# B&R Automation Studio project TD52 (part 98)

#### MsgEXCyclic.st
```iecst
(*******************************************************************************
MsgEX	 			 alarms, messages MM_EX

This code is confidential and proprietary to the INNIO Company.
It may not be used in any form, or reproduced in any manner,
without written permission of the INNIO Company.
Copyright, INNIO Company, 2025

Customized modifications: -
------------------------

History:
-------
V3.99.0	04.06.2012	lettenb.	new
		20.03.2013				para.cleanup
		23.04.2013				reset OUT_EX.tEX2AB.bGnlWarning added
		16.05.2013				3349,3580,3581,3582 added from V3.30.x
		23.05.2013				2847,2848 added
		24.05.2013				reset OUT_xx.txx2AB.bGnlTripx changed
		28.05.2013				2622,2623 for 424tstc added
		04.06.2013				1163,1171 var.names changed(EGbHE -> EGaTC)
								1172 limit var.changed, bugfix
		23.07.2013				2576,2577 enabled if sensor active
		17.01.2014				3366,3417 added, 1165 disabled (exh.gas scav. after engine stop)
V4.00.0	26.02.2014				logger entries added
V4.00.1	09.04.2014				3417 disabled for engines without EGScav
V4.00.2	14.05.2014				1172 KK_AUF AND BTRB added, ton 0s->120s (anforderung requisition/poppe,a_v3500)
		27.05.2014				1172 KK_AUF -> OUT_EX.EG_BoVaOpened (universal for combi valves)
		23.06.2014				2098 logic in case of Para.bSel_EGVa_Combi separated, bugfix
		08.08.2014				3417 IN_EX.bMsg1078 added, to avoid alarm in case of signal failure
V4.00.3 21.01.2015 lettenb.		2655-2664 added(Gen2 engine controller)
		11.02.2015				1165,3366 prepared FOR blackstart,
								3510 logic corr.(bugfix)
								1163 enable with IN_VE.tPB2MM.bSys_Run
								1273-1280 added
V4.03.0 27.07.2015 Plattner		2743 - 2748 & 3397 added. differential pressure exhaust gas cooler and filter limits and msf
								1288 - 1291 added operations message from CO2 flap
        05.08.2015 Stary        added 3394+3395 & 3490+3491
		14.07.2016 lettenb.		3491 xGR_MAXR_T_EGaHE2_LimHi_Warn: Ai+Para changed, 3394,3395,3490,3491 TON 0->2s, double 3395 removed, bugfix
		22.09.2016 lettenb.		1291 NOT added, bugfix
		04.10.2016				2793 added, FC monitoring
		09.02.2017				3417 trip prio corr. 3 -> 4
V4.05.0 21.03.2017 lettenb.     3100 disabled for 920, SWAT920/2
		28.06.2017				2847,2848 N2 gas valve open/closed changed, bugfix
		12.07.2017 Messner		A2315, W2468, W2469 added and W3417 para added
		09.10.2017 Weitzer		3100 enable for 920 again! Increase time delay from 2s TO 120s. SWAT920/x
		02.08.2017				2847,2848 N2 valves open/closed changed, synch.acc.VIS, bu09
		04.12.2017 Messner		Oxidation catalyst added
								Old KAT Disabled: A1045, A1069; W1161, W1162,  W1169, W1170, W1174, W2112;
								New OXIcat Added: A2319, A2320; W2494, W2495, W2496, W2497, W2498, W2499, W2500;
		22.05.2017	TinelloM	SCR deleted
		20.12.2017	lettenb.	A3397 prio: 4->3, bugfix
		02.01.2017	lettenb.	3417 disabled for 920 with common gas train(main and prechamber)(not for ACEA,sky,rosenheim,stapelfeld)
		18.01.2018				2310,2311,2312,2313 added, 1171,2546,2547:Para.rT_EGaTC_HyHi removed(burkhart)
		22.01.2018	lettenb.	1163,1164,2793 bSys_Run -> bParaSetupOk to avoid message at plc startup
V4.05.1 19.03.2018	lettenb.    2320,2500 delay 1s added to avoid alarm with siganl failure, bugfix
V4.07.0 26.04.2018	lettenb.	9215 added, 1165 enabled for BR9, 3366 disabled for BR9, SWAT920/5
		08.10.2018	lettenb.	3214, :bOMSS... removed, signal failure active in stop-mode
		31.10.2018	lettenb.	2321,2322 added, (burkhart)
		03.12.2018	lettenb.	1165,3366,1279,1280 NoScavFan added, bugfix for option N2 scav.without scav.fan
		14.01.2019	Schmid		A2340+W9249 added, W2498+W2497 deactivated, "exhaust gas pressure fast" fully replaces "OXIcat inlet pressure fast"
		18.03.2019	lettenb.	2497,2498 cleanup unused code
		13.06.2019	lettenb.	1171,2310,2311,2546,2547: MM2VIS.bMsg2312/2313/2322 added to avoid hi-alarm with MS, bugfix
		03.10.2019	lettenb.	9310 added, 2319 disabled, OXIcat monitoring, bu
V4.09.0	02.08.2019	lettenb.	2337,2338,9305-9308: temperature exhaust gas pressure relief valve 1/2 added
		13.07.2020	lettenb.	2496 time delay 60s added, bu
V4.11.0 04.03.2021	lettenb.	9347,9348 added, exhaust gas flap monitoring
V4.12.0	19.12.2022	Perktold	added comments for sr-code (EN 13849-1 / 4.6.3) for A1092,A2315 & W3528
V4.13.0	19.10.2023	Heim Markus	add A2374 (defined as safety critical no remote reset possible (riskclass 10)
V4.14.0	16.10.2024	VighM		W9249 set by bad signal quality, delay cleanup.
V4.14.0	06.11.2024	Theobald	At alarm 1092 only temperature sensor cause trip while the engine is running and at alarm 3366 there is no trip during engine operation.
		25.11.2024	Bacci		T6 Start procedure with purge start (2024-219): scavenging fan removal
V4.25.0	10.07.2025	Tinello	 	SafetyPLC: Disabled W3528 in case of Safety gas backpressure monitoring active

Instructions for use:
--------------------
1) declare alarm with FUNCTION block "Alm"
	declare buffert alarm bit bMsg<message number>

2) use template to create a new alarm,
   substitue 0000 by alarm number and make settings:

	xMsg0000.Enable		:=	TRUE;		enable/disable alarm
	xMsg0000.Set		:=	FALSE;		alarm set condition
	xMsg0000.PT			:=	T#0s;		alarm delay time
	xMsg0000.Prio		:=	1;			alarm priority: 1-3 = trip, 4 = warning
	xMsg0000.RiskClass	:=	3;			risk class for remote alarm reset
	xMsg0000.Reset		:=	FALSE;		FALSE: for all standard alarms	prio 1,2,3 and warnings prio 4
										TRUE : for autoreset alarms

	bMsg0000			:=	xMsg0000.Q;	connect buffert alarm bit for VIS and control
	bMsg0000_Test		:=	xMsg0000.Test; alarm bypass active

3)  expand INIT

4)	include datapoint into OPC configuration for vis

Outstandings:
------------
logic FOR alarm 2622,2623 (424)
W exhaust gas scavenging before next start
(*******************************************************************************)
PROGRAM _CYCLIC

	(* reset general trip *)
	OUT_EX.tEX2AB.bGnlTrip1		:=	FALSE;
	OUT_EX.tEX2AB.bGnlTrip2		:=	FALSE;
	OUT_EX.tEX2AB.bGnlTrip3		:=	FALSE;
	OUT_EX.tEX2AB.bGnlWarning	:=	FALSE;
	OUT_EX.tEX2AB.bTriptype1	:=	FALSE;
	OUT_EX.tEX2AB.bTriptype2	:=	FALSE;
	OUT_EX.tEX2AB.bTriptype3	:=	FALSE;

	(*-------------------------------------------------------------------------*)
	(* A1045 catalyst temperature high (W1174) *) (* Disabled - OXIcat *)
	xMsg1045.Enable	   := FALSE;
	xMsg1045.Set	   := FALSE;
	xMsg1045.PT		   := T#0s;
	xMsg1045.Prio 	   := 2;
	xMsg1045.RiskClass := 4;
	xMsg1045.Reset     := FALSE;
	xMsg1045();
	MM2VIS.bMsg1045    := xMsg1045.Q;

	(* A1046 exhaust gas flap failure (--> W2098) *)
	xMsg1046.Enable	   := FALSE;
	xMsg1046.Set 	   := FALSE;
	xMsg1046.PT		   := T#0s;
	xMsg1046.Prio 	   := 3;
	xMsg1046.RiskClass := 3;
	xMsg1046.Reset     := FALSE;
	xMsg1046();
	MM2VIS.bMsg1046    := xMsg1046.Q;

	(* A1069 catalyst temperature signal failure (W2112) *) (* Disabled - OXIcat *)
	xMsg1069.Enable	   := FALSE;
	xMsg1069.Set 	   := FALSE;
	xMsg1069.PT		   := T#0s;
	xMsg1069.Prio 	   := 3;
	xMsg1069.RiskClass := 2;
	xMsg1069.Reset     := FALSE;
	xMsg1069();
	MM2VIS.bMsg1069    := xMsg1069.Q;

	(********************************************************************************************************************
	Safety-related application software source code (EN 13849-1 / 4.6.3): BEGIN
	*********************************************************************************************************************)

	(* A1092 exhaust gas scavenging valve failure *)
	xMsg1092.Enable	   := TRUE;
	xMsg1092.Set 	   := (T1_STSPKL AND NOT IN_EX.tEng_Run.Do) OR T2_STSPKL;
	xMsg1092.PT		   := T#0s;
	xMsg1092.Prio 	   := 2;
	xMsg1092.RiskClass := 10;
	xMsg1092.Reset     := FALSE;
	xMsg1092();
	MM2VIS.bMsg1092    := xMsg1092.Q;

	(********************************************************************************************************************
	Safety-related application software source code (EN 13849-1 / 4.6.3): END
	*********************************************************************************************************************)

	(* A1104 plate temperature heat exchanger high *)
	xGR_MAXR_T_PlateHE_LimHiHi(In:= IN_EX.tT_PlateHE.Ai, Gw:= Para.rT_PlateHE_LimHiHi, Hy:= Para.rT_PlateHE_HyHi);

	xMsg1104.Enable	   := Para.bT_PlateHE_Active;
	xMsg1104.Set 	   := xGR_MAXR_T_PlateHE_LimHiHi.Q AND IN_EX.tPB2MM.bParaSetupOk AND NOT MM2VIS.bMsg2113;
	xMsg1104.PT		   := T#2s;
	xMsg1104.Prio 	   := 3;
	xMsg1104.RiskClass := 4;
	xMsg1104.Reset     := FALSE;
	xMsg1104();
	MM2VIS.bMsg1104    := xMsg1104.Q;

	(* A1106 plate temperature heat exchanger signal failure(--> W2113) *)
	xMsg1106.Enable	   := Para.bT_PlateHE_Active AND FALSE;
	xMsg1106.Set 	   := NOT IN_EX.tT_PlateHE.GoodQual;
	xMsg1106.PT		   := T#0s;
	xMsg1106.Prio 	   := 3;
	xMsg1106.RiskClass := 4;
	xMsg1106.Reset     := FALSE;
	xMsg1106();
	MM2VIS.bMsg1106    := xMsg1106.Q;

	(* W1161 exhaust gas temperature before catalyst signal failure *) (* Disabled - OXIcat *)
	xMsg1161.Enable	   := FALSE;
	xMsg1161.Set 	   := FALSE;
	xMsg1161.PT		   := T#0s;
	xMsg1161.Prio 	   := 4;
	xMsg1161.RiskClass := 4;
	xMsg1161.Reset     := FALSE;
	xMsg1161();
	MM2VIS.bMsg1161    := xMsg1161.Q;

	(* W1162 exhaust gas temperature after catalyst signal failure *) (* Disabled - OXIcat *)
	xMsg1162.Enable	   := FALSE;
	xMsg1162.Set 	   := FALSE;
	xMsg1162.PT		   := T#0s;
	xMsg1162.Prio 	   := 4;
	xMsg1162.RiskClass := 4;
	xMsg1162.Reset     := FALSE;
	xMsg1162();
	MM2VIS.bMsg1162    := xMsg1162.Q;

	(* W1163 (A2322) exhaust gas temperature after turbo charger signal failure *)
	xMsg1163.Enable	   := Para.bT_EGaTC_Active AND IN_EX.tPB2MM.bParaSetupOk;
	xMsg1163.Set 	   := NOT IN_EX.tT_EGaTC.GoodQual AND NOT Para.bT_EGaLPTC_HiTrip;
	xMsg1163.PT		   := T#0s;
	xMsg1163.Prio 	   := 4;
	xMsg1163.RiskClass := 4;
	xMsg1163.Reset     := FALSE;
	xMsg1163();
	MM2VIS.bMsg1163    := xMsg1163.Q;

	(* W1164 exhaust gas temperature after heat exchanger signal failure *)
	xMsg1164.Enable	   := Para.bT_EGaHE_Active AND IN_EX.tPB2MM.bParaSetupOk;
	xMsg1164.Set 	   := NOT IN_EX.tT_EGaHE.GoodQual;
	xMsg1164.PT		   := T#0s;
	xMsg1164.Prio 	   := 4;
	xMsg1164.RiskClass := 4;
	xMsg1164.Reset     := FALSE;
	xMsg1164();
	MM2VIS.bMsg1164    := xMsg1164.Q;

   (* W1165 exhaust gas scavenging fan failure (A3366) *)
	xTOF_EngDemEPS(IN:= IN_EX.bEng_Dem_EPS AND NOT IN_EX.tGCB_On.Di, PT:= T#60s);
	bNoMon4BlackStart := xTOF_EngDemEPS.Q AND IN_EX.bEng_Dem_EPS; //T14

	xMsg1165.Enable	   := xEngType.Type9;//SWAT920/5
	xMsg1165.Set 	   :=	OUT_EX.tScavFanCoOn.Do
					AND NOT bNoMon4BlackStart
					AND(   (NOT xEngType.Type9 AND NOT IN_EX.tScavFanOp.Di AND NOT NoScavFan)
						OR (    xEngType.Type9 AND    (IN_EX.tScavFanFC_P_Lo.Di OR NOT IN_EX.tScavFanFC_Rdy.Di)));
	xMsg1165.PT		   := T#10s;
	xMsg1165.Prio 	   := 4;
	xMsg1165.RiskClass := 4;
	xMsg1165.Reset     := FALSE;
	xMsg1165();
	MM2VIS.bMsg1165	   := xMsg1165.Q;
	OUT_EX.bMsg1165	   := xMsg1165.Q;//SWAT920/5

	(* W1169 exhaust gas temperature before catalyst high *) (* Disabled - OXIcat *)
	xMsg1169.Enable	   := FALSE;
	xMsg1169.Set 	   := FALSE;
	xMsg1169.PT		   := T#2s;
	xMsg1169.Prio 	   := 4;
	xMsg1169.RiskClass := 4;
	xMsg1169.Reset     := FALSE;
	xMsg1169();
	MM2VIS.bMsg1169    := xMsg1169.Q;

	(* W1170 exhaust gas temperature after catalyst high *) (* Disabled - OXIcat *)
	xMsg1170.Enable	   := FALSE;
	xMsg1170.Set 	   := FALSE;
	xMsg1170.PT		   := T#2s;
	xMsg1170.Prio 	   := 4;
	xMsg1170.RiskClass := 4;
	xMsg1170.Reset     := FALSE;
	xMsg1170();
	MM2VIS.bMsg1170    := xMsg1170.Q;

	(* W1171 (A2321) exhaust gas temperature after turbo charger high *)
	xGR_MAXR_T_EGaTC_LimHi(In:= IN_EX.tT_EGaTC.Ai, Gw:= Para.rT_EGaTC_LimHi, Hy:= 5.0);

	xMsg1171.Enable	   := Para.bT_EGaTC_Active;
	xMsg1171.Set 	   := xGR_MAXR_T_EGaTC_LimHi.Q AND IN_EX.tPB2MM.bParaSetupOk AND NOT MM2VIS.bMsg1163 AND NOT MM2VIS.bMsg2322;
	xMsg1171.PT		   := T#2s;
	xMsg1171.Prio 	   := 4;
	xMsg1171.RiskClass := 4;
	xMsg1171.Reset     := FALSE;
	xMsg1171();
	MM2VIS.bMsg1171    := xMsg1171.Q;

	(* W1172 exhaust gas temperature after heat exchanger high *)
	xGR_MAXR_T_EGaHE_LimHi(In:= IN_EX.tT_EGaHE.Ai, Gw:= Para.rT_EGaHE_LimHi, Hy:= Para.rT_EGaHE_HyHi);

	xMsg1172.Enable	   := Para.bT_EGaHE_Active;
	xMsg1172.Set 	   := xGR_MAXR_T_EGaHE_LimHi.Q AND IN_EX.tPB2MM.bParaSetupOk AND NOT MM2VIS.bMsg1164
					  AND OUT_EX.bEG_BoVaOpened AND IN_EX.tEng_Run.Do;
	xMsg1172.PT		   := T#120s;
	xMsg1172.Prio 	   := 4;
	xMsg1172.RiskClass := 4;
	xMsg1172.Reset     := FALSE;
	xMsg1172();
	MM2VIS.bMsg1172    := xMsg1172.Q;

	(* W1173 plate temperature heat exchanger high *)
	xGR_MAXR_T_PlateHE_LimHi(In:= IN_EX.tT_PlateHE.Ai, Gw:= Para.rT_PlateHE_LimHi, Hy:= Para.rT_PlateHE_HyHi);

	xMsg1173.Enable	   := Para.bT_PlateHE_Active;
	xMsg1173.Set 	   := xGR_MAXR_T_PlateHE_LimHi.Q AND IN_EX.tPB2MM.bParaSetupOk AND NOT MM2VIS.bMsg2113;
	xMsg1173.PT		   := T#2s;
	xMsg1173.Prio 	   := 4;
	xMsg1173.RiskClass := 4;
	xMsg1173.Reset     := FALSE;
	xMsg1173();
	MM2VIS.bMsg1173    := xMsg1173.Q;

	(* W1174 catalyst temperatur high (A1045) *) (* Disabled - OXIcat *)
	xMsg1174.Enable	   := FALSE;
	xMsg1174.Set 	   := FALSE;
	xMsg1174.PT		   := T#2s;
	xMsg1174.Prio 	   := 4;
	xMsg1174.RiskClass := 4;
	xMsg1174.Reset     := FALSE;
	xMsg1174();
	MM2VIS.bMsg1174    := xMsg1174.Q;

	(* W2098 exhaust gas flap failure *)
	IF Para.bSel_EGVa_Combi THEN
		xTON_2098a(IN:= (NOT IN_EX.tEG_ByVaOpened.Di AND NOT IN_EX.tEG_ByVaClosed.Di AND(B_BKAUF OR B_BKZU)), PT:= T#35s);
	ELSE
		xTON_2098a(IN:= (NOT IN_EX.tEG_ByVaOpened.Di AND NOT IN_EX.tEG_ByVaClosed.Di AND(B_BKAUF OR B_BKZU))
					 OR (NOT IN_EX.tEG_BoVaOpened.Di AND NOT IN_EX.tEG_BoVaClosed.Di AND(B_KKAUF OR B_KKZU)), PT:= T#35s);
	END_IF;
	xTON_2098b(IN:=  NOT IN_EX.tEG_BoVaFailure.Di OR NOT IN_EX.tEG_ByVaFailure.Di, PT:= T#2s);

	xMsg2098.Enable	   := TRUE;
	xMsg2098.Set 	   := xTON_2098a.Q OR xTON_2098b.Q OR (NOT Para.bSel_EGVa_Combi AND NOT IN_EX.tEG_ByVaOpened.Di AND NOT IN_EX.tEG_BoVaOpened.Di);
	xMsg2098.PT		   := T#0s;
	xMsg2098.Prio 	   := 4;
	xMsg2098.RiskClass := 4;
	xMsg2098.Reset     := FALSE;
	xMsg2098();
	MM2VIS.bMsg2098    := xMsg2098.Q;

	(* W2112 catalyst temperature signal failure (A1069) *) (* Disabled - OXIcat *)
	xMsg2112.Enable	   := FALSE;
	xMsg2112.Set 	   := FALSE;
	xMsg2112.PT		   := T#0s;
	xMsg2112.Prio 	   := 4;
	xMsg2112.RiskClass := 4;
	xMsg2112.Reset     := FALSE;
	xMsg2112();
	MM2VIS.bMsg2112    := xMsg2112.Q;

	(* W2113 plate temperature heat exchanger signal failure (A1106) *)
	xMsg2113.Enable	   := Para.bT_PlateHE_Active;
	xMsg2113.Set 	   := NOT IN_EX.tT_PlateHE.GoodQual;
	xMsg2113.PT		   := T#0s;
	xMsg2113.Prio 	   := 4;
	xMsg2113.RiskClass := 4;
	xMsg2113.Reset     := FALSE;
	xMsg2113();
	MM2VIS.bMsg2113    := xMsg2113.Q;

	(* A2310 (W2546) exhaust gas temperature after low pressure turbo charger A high *)(* M.02-TI-168, M.02-TI-001 *)
	xMsg2310.Enable	   := Para.bT_EGaLPTC_A_Active AND Para.bT_EGaLPTC_HiTrip;
	xMsg2310.Set 	   := IN_EX.tPB2MM.bParaSetupOk AND (IN_EX.tT_EGaLPTC_A.Ai > Para.rT_EGaTC_LimHiHi) AND NOT MM2VIS.bMsg2312;
	xMsg2310.PT		   := Para.tiEGaTC_LimHiHi;
	xMsg2310.Prio 	   := 2;
	xMsg2310.RiskClass := 4;
	xMsg2310.Reset     := FALSE;
	xMsg2310();
	MM2VIS.bMsg2310    := xMsg2310.Q;

	(* A2311 (W2547) exhaust gas temperature after low pressure turbo charger B high *)(* M.02-TI-268, M.02-TI-002 *)
	xMsg2311.Enable	   := Para.bT_EGaLPTC_B_Active AND Para.bT_EGaLPTC_HiTrip;
	xMsg2311.Set 	   := IN_EX.tPB2MM.bParaSetupOk AND (IN_EX.tT_EGaLPTC_B.Ai > Para.rT_EGaTC_LimHiHi) AND NOT MM2VIS.bMsg2313;
	xMsg2311.PT		   := Para.tiEGaTC_LimHiHi;
	xMsg2311.Prio 	   := 2;
	xMsg2311.RiskClass := 4;
	xMsg2311.Reset     := FALSE;
	xMsg2311();
	MM2VIS.bMsg2311    := xMsg2311.Q;

	(* A2312 (W2549) exhaust gas temperature after low pressure turbo charger A signal failure *)(* M.02-TI-168, M.02-TI-001 *)
	xMsg2312.Enable	   := Para.bT_EGaLPTC_A_Active AND Para.bT_EGaLPTC_HiTrip;
	xMsg2312.Set 	   := IN_EX.tPB2MM.bParaSetupOk AND NOT IN_EX.tT_EGaLPTC_A.GoodQual;
	xMsg2312.PT		   := T#0s;
	xMsg2312.Prio 	   := 2;
	xMsg2312.RiskClass := 4;
	xMsg2312.Reset     := FALSE;
	xMsg2312();
	MM2VIS.bMsg2312    := xMsg2312.Q;

	(* A2313 (W2551) exhaust gas temperature after low pressure turbo charger B signal failure *)(* M.02-TI-268, M.02-TI-002 *)
	xMsg2313.Enable	   := Para.bT_EGaLPTC_B_Active AND Para.bT_EGaLPTC_HiTrip;
	xMsg2313.Set 	   := IN_EX.tPB2MM.bParaSetupOk AND NOT IN_EX.tT_EGaLPTC_B.GoodQual;
	xMsg2313.PT		   := T#0s;
	xMsg2313.Prio 	   := 2;
	xMsg2313.RiskClass := 4;
	xMsg2313.Reset     := FALSE;
	xMsg2313();
	MM2VIS.bMsg2313    := xMsg2313.Q;

	(********************************************************************************************************************
	Safety-related application software source code (EN 13849-1 / 4.6.3): BEGIN
	*********************************************************************************************************************)

	(* A2315 air temperature before exhaust gas scavening valve maximum *)
	xMsg2315.Enable	   := Para.bT_bScavValve_Active;
	xMsg2315.Set 	   := IN_EX.tPB2MM.bParaSetupOk AND  IN_EX.tT_bScavValve.GoodQual
													AND (IN_EX.rN_EngAct > 0)
													AND (IN_EX.tT_bScavValve.Ai > Para.rT_bScavValve_LimHi);
	xMsg2315.PT		   := T#2s;
	xMsg2315.Prio 	   := 2;
	xMsg2315.RiskClass := 10;
	xMsg2315.Reset     := FALSE;
	xMsg2315();
	MM2VIS.bMsg2315    := xMsg2315.Q;

	(********************************************************************************************************************
	Safety-related application software source code (EN 13849-1 / 4.6.3): END
	*********************************************************************************************************************)

	(* A2319 OXIcat Outlet temperature measurement signal failure *)(* W9310 *)
	xMsg2319.Enable	   := Para.bOXIcat_Exist
					  AND Para.bT_OXIcat_Out_Exist
					  AND FALSE;
	xMsg2319.Set 	   := NOT IN_EX.tT_EGaCat.GoodQual
					  AND (IN_EX.rN_EngAct > 0);
	xMsg2319.PT		   := T#2s;
	xMsg2319.Prio 	   := 3;
	xMsg2319.RiskClass := 4;
	xMsg2319.Reset     := FALSE;
	xMsg2319();
	MM2VIS.bMsg2319    := xMsg2319.Q;

	(* A2320 OXIcat Outlet temperature maximum *)
	xMsg2320.Enable	   := Para.bOXIcat_Exist
					  AND Para.bT_OXIcat_Out_Exist;
	xMsg2320.Set 	   := IN_EX.tT_EGaCat.Ai >= Para.rT_OXIcat_Out_HiHi
					  AND (IN_EX.rN_EngAct > 0)
					  AND IN_EX.tT_EGaCat.GoodQual;
	xMsg2320.PT		   := T#1s;
	xMsg2320.Prio 	   := 2;
	xMsg2320.RiskClass := 4;
	xMsg2320.Reset     := FALSE;
	xMsg2320();
	MM2VIS.bMsg2320    := xMsg2320.Q;

	(* A2321 (W1171) exhaust gas temperature after turbo charger high *)(* M.02-TI-001 *)
	xMsg2321.Enable	   := Para.bT_EGaTC_Active AND Para.bT_EGaLPTC_HiTrip;
	xMsg2321.Set 	   := IN_EX.tPB2MM.bParaSetupOk AND (IN_EX.tT_EGaTC.Ai > Para.rT_EGaTC_LimHiHi) AND NOT MM2VIS.bMsg2322;
	xMsg2321.PT		   := Para.tiEGaTC_LimHiHi;
	xMsg2321.Prio 	   := 2;
	xMsg2321.RiskClass := 4;
	xMsg2321.Reset     := FALSE;
	xMsg2321();
	MM2VIS.bMsg2321    := xMsg2321.Q;

	(* A2322 (W1163) exhaust gas temperature after turbo charger signal failure *)(* M.02-TI-001 *)
	xMsg2322.Enable	   := Para.bT_EGaTC_Active AND Para.bT_EGaLPTC_HiTrip;
	xMsg2322.Set 	   := IN_EX.tPB2MM.bParaSetupOk AND NOT IN_EX.tT_EGaTC.GoodQual;
	xMsg2322.PT		   := T#0s;
	xMsg2322.Prio 	   := 2;
	xMsg2322.RiskClass := 4;
	xMsg2322.Reset     := FALSE;
	xMsg2322();
	MM2VIS.bMsg2322    := xMsg2322.Q;

	(********************************************************************************************************************
	Safety-related application software source code (EN 13849-1 / 4.6.3): BEGIN
	*********************************************************************************************************************)

	(* A2337 (W9305) temperature high exhaust gas pressure relief valve 1 *)(* P.02-TI-039 *)
	xMsg2337.Enable	   := Para.bT_EG_PrReliefVa1_Active;
	xMsg2337.Set 	   := IN_EX.tPB2MM.bParaSetupOk AND(IN_EX.tT_EG_PrReliefVa1.Ai > Para.rT_EG_PrReliefVa_LimHiHi) AND NOT MM2VIS.bMsg9307;
	xMsg2337.PT		   := T#2s;
	xMsg2337.Prio 	   := 3;
	xMsg2337.RiskClass := 10;
	xMsg2337.Reset     := FALSE;
	xMsg2337();
	MM2VIS.bMsg2337    := xMsg2337.Q;

	(* A2338 (W9306) temperature high exhaust gas pressure relief valve 2 *)(* P.02-TI-040 *)
	xMsg2338.Enable	   := Para.bT_EG_PrReliefVa2_Active;
	xMsg2338.Set 	   := IN_EX.tPB2MM.bParaSetupOk AND(IN_EX.tT_EG_PrReliefVa2.Ai > Para.rT_EG_PrReliefVa_LimHiHi) AND NOT MM2VIS.bMsg9308;
	xMsg2338.PT		   := T#2s;
	xMsg2338.Prio 	   := 3;
	xMsg2338.RiskClass := 10;
	xMsg2338.Reset     := FALSE;
	xMsg2338();
	MM2VIS.bMsg2338    := xMsg2338.Q;

	(********************************************************************************************************************
	Safety-related application software source code (EN 13849-1 / 4.6.3): END
	*********************************************************************************************************************)

	(* A2340 Exhaust gas pressure fast maximum (W2498) *)
	xMsg2340.Enable	   := Para.bPr_OXIcat_In_Fast_Exist;
	xMsg2340.Set 	   := bPr_EG_Deflag_Fast
					  AND NOT xTOF_Pr_EG_Deflag_Fast.Q
					  AND ((IN_EX.rN_EngAct > 0) OR IN_EX.bEng_Start) // Prevents continuous setting of the alarm, while bPr_EG_Deflag_Fast remains active
					  AND NOT MM2VIS.bMsg9249;
	xMsg2340.PT		   := T#0s;
	xMsg2340.Prio 	   := 2;
	xMsg2340.RiskClass := 4;
	xMsg2340.Reset     := FALSE;
	xMsg2340();
	MM2VIS.bMsg2340    := xMsg2340.Q;

	(********************************************************************************************************************
	Safety-related application software source code (EN 13849-1 / 4.6.3): BEGIN
	*********************************************************************************************************************)

	(* A2374 Bursting disc triggered (P.02-GS-001/P.02-GS-002)*)
	xMsg2374.Enable	   := IN_EX.tPB2MM.bParaSetupOk;
	xMsg2374.Set 	   := NOT IN_EX.tBurstingDisk1_Ok.Di
					   OR NOT IN_EX.tBurstingDisk2_Ok.Di;
	xMsg2374.PT		   := T#0s;
	xMsg2374.Prio 	   := 2;
	xMsg2374.RiskClass := 10;
	xMsg2374.Reset     := FALSE;
	xMsg2374();
	MM2VIS.bMsg2374    := xMsg2374.Q;

	(********************************************************************************************************************
	Safety-related application software source code (EN 13849-1 / 4.6.3): END
	*********************************************************************************************************************)

	(* W2468 air temperature before exhaust gas scavening valve signal failure *)
	xMsg2468.Enable	   := Para.bT_bScavValve_Active;
	xMsg2468.Set 	   := IN_EX.tPB2MM.bParaSetupOk AND NOT IN_EX.tT_bScavValve.GoodQual;
	xMsg2468.PT		   := T#0s;
	xMsg2468.Prio 	   := 4;
	xMsg2468.RiskClass := 4;
	xMsg2468.Reset     := FALSE;
	xMsg2468();
	MM2VIS.bMsg2468    := xMsg2468.Q;

	(* W2469 air temperature before exhaust gas scavening valve plausibility check *)
	xMsg2469.Enable	   := Para.bT_bScavValve_Active AND FALSE;//SWAT920/5
	xMsg2469.Set 	   := IN_EX.tPB2MM.bParaSetupOk AND bT_bScavValve_PcheckFail;
	xMsg2469.PT		   := T#0s;
	xMsg2469.Prio 	   := 4;
	xMsg2469.RiskClass := 4;
	xMsg2469.Reset     := FALSE;
	xMsg2469();
	MM2VIS.bMsg2469    := xMsg2469.Q;

	(* W2494 OXIcat Inlet pressure measurement signal failure *)
	xMsg2494.Enable	   := Para.bOXIcat_Exist
					  AND Para.bPr_OXIcat_In_Exist;
	xMsg2494.Set 	   := NOT IN_EX.tPr_OXIcat_In.GoodQual
					  AND (IN_EX.rP_Act_Norm_Filt >= 0.50);
	xMsg2494.PT		   := T#60s;
	xMsg2494.Prio 	   := 4;
	xMsg2494.RiskClass := 4;
	xMsg2494.Reset     := FALSE;
	xMsg2494();
	MM2VIS.bMsg2494    := xMsg2494.Q;

	(* W2495 OXIcat Outlet pressure measurement signal failure *)
	xMsg2495.Enable	   := Para.bOXIcat_Exist
					  AND Para.bPr_OXIcat_Out_Exist;
	xMsg2495.Set 	   := NOT IN_EX.tPr_OXIcat_Out.GoodQual
					  AND (IN_EX.rP_Act_Norm_Filt >= 0.50);
	xMsg2495.PT		   := T#60s;
	xMsg2495.Prio 	   := 4;
	xMsg2495.RiskClass := 4;
	xMsg2495.Reset     := FALSE;
	xMsg2495();
	MM2VIS.bMsg2495    := xMsg2495.Q;

	(* W2496 OXIcat Differential pressure minimum *)
	xMsg2496.Enable	   := Para.bOXIcat_Exist
					  AND Para.bPr_OXIcat_In_Exist
					  AND Para.bPr_OXIcat_Out_Exist;
	xMsg2496.Set 	   := MM2VIS.rPr_OXIcat_Diff <= Para.rPR_OXIcat_Diff_Hi
					  AND (IN_EX.rP_Act_Norm_Filt >= 0.50)
					  AND IN_EX.tPr_OXIcat_In.GoodQual
					  AND IN_EX.tPr_OXIcat_Out.GoodQual;
	xMsg2496.PT		   := T#60s;
	xMsg2496.Prio 	   := 4;
	xMsg2496.RiskClass := 4;
	xMsg2496.Reset     := FALSE;
	xMsg2496();
	MM2VIS.bMsg2496    := xMsg2496.Q;

	(* W2497 OXIcat Exhaust gas inlet pressure fast measurement signal failure *)
	xMsg2497.Enable	   := FALSE;	(*v4.07*)
	xMsg2497.Set 	   := FALSE;
	xMsg2497.PT		   := T#60s;
	xMsg2497.Prio 	   := 4;
	xMsg2497.RiskClass := 4;
	xMsg2497.Reset     := FALSE;
	xMsg2497();
	MM2VIS.bMsg2497    := xMsg2497.Q;

	(* W2498 OXIcat Exhaust gas inlet pressure fast maximum *)
	xMsg2498.Enable	   := FALSE;	(*v4.07*)
	xMsg2498.Set 	   := FALSE;
	xMsg2498.PT		   := T#0s;
	xMsg2498.Prio 	   := 4;
	xMsg2498.RiskClass := 4;
	xMsg2498.Reset     := FALSE;
	xMsg2498();
	MM2VIS.bMsg2498    := xMsg2498.Q;

	(* W2499 OXIcat Inlet temperature measurement signal *)
	xMsg2499.Enable	   := Para.bOXIcat_Exist
					  AND Para.bT_OXIcat_In_Exist;
	xMsg2499.Set 	   := NOT IN_EX.tT_EGbCat.GoodQual
					  AND (IN_EX.rN_EngAct > 0);
	xMsg2499.PT		   := T#60s;
	xMsg2499.Prio 	   := 4;
	xMsg2499.RiskClass := 4;
	xMsg2499.Reset     := FALSE;
	xMsg2499();
	MM2VIS.bMsg2499    := xMsg2499.Q;

	(* W2500 OXIcat Inlet temperature high *)
	xMsg2500.Enable	   := Para.bOXIcat_Exist
					  AND Para.bT_OXIcat_In_Exist;
	xMsg2500.Set 	   := IN_EX.tT_EGbCat.Ai >= Para.rT_OXIcat_In_Hi
					  AND (IN_EX.rN_EngAct > 0)
					  AND IN_EX.tT_EGbCat.GoodQual;
	xMsg2500.PT		   := T#1s;
	xMsg2500.Prio 	   := 4;
	xMsg2500.RiskClass := 4;
	xMsg2500.Reset     := FALSE;
	xMsg2500();
	MM2VIS.bMsg2500    := xMsg2500.Q;

	(* W2546 (A2310) exhaust gas temperature after low pressure turbo charger A high *)(* M.02-TI-168, M.02-TI-001 *)
	xGR_MAXR_T_EGaLPTC_A_LimHi(In:= IN_EX.tT_EGaLPTC_A.Ai, Gw:= Para.rT_EGaTC_LimHi, Hy:= 5.0);

	xMsg2546.Enable	   := Para.bT_EGaLPTC_A_Active;
	xMsg2546.Set 	   := IN_EX.tPB2MM.bParaSetupOk AND xGR_MAXR_T_EGaLPTC_A_LimHi.Q AND Para.bT_EGaLPTC_A_Active AND NOT MM2VIS.bMsg2549 AND NOT MM2VIS.bMsg2312;
	xMsg2546.PT		   := T#2s;
	xMsg2546.Prio 	   := 4;
	xMsg2546.RiskClass := 4;
	xMsg2546.Reset     := FALSE;
	xMsg2546();
	MM2VIS.bMsg2546    := xMsg2546.Q;

	(* W2547 (A2311) exhaust gas temperature after low pressure turbo charger B high *)(* M.02-TI-268, M.02-TI-002 *)
	xGR_MAXR_T_EGaLPTC_B_LimHi(In:= IN_EX.tT_EGaLPTC_B.Ai, Gw:= Para.rT_EGaTC_LimHi, Hy:= 5.0);

	xMsg2547.Enable	   := Para.bT_EGaLPTC_B_Active;
	xMsg2547.Set 	   := IN_EX.tPB2MM.bParaSetupOk AND xGR_MAXR_T_EGaLPTC_B_LimHi.Q AND Para.bT_EGaLPTC_B_Active AND NOT MM2VIS.bMsg2551 AND NOT MM2VIS.bMsg2313;
	xMsg2547.PT		   := T#2s;
	xMsg2547.Prio 	   := 4;
	xMsg2547.RiskClass := 4;
	xMsg2547.Reset     := FALSE;
	xMsg2547();
	MM2VIS.bMsg2547    := xMsg2547.Q;

	(* W2549 exhaust gas temperature after low pressure turbo charger A signal failure *)(* M.02-TI-168, M.02-TI-001 *)
	xMsg2549.Enable	   := Para.bT_EGaLPTC_A_Active AND NOT Para.bT_EGaLPTC_HiTrip;
	xMsg2549.Set 	   := IN_EX.tPB2MM.bParaSetupOk AND NOT IN_EX.tT_EGaLPTC_A.GoodQual;
	xMsg2549.PT		   := T#0s;
	xMsg2549.Prio 	   := 4;
	xMsg2549.RiskClass := 4;
	xMsg2549.Reset     := FALSE;
	xMsg2549();
	MM2VIS.bMsg2549    := xMsg2549.Q;

	(* W2551 exhaust gas temperature after low pressure turbo charger B signal failure *)(* M.02-TI-268, M.02-TI-002 *)
	xMsg2551.Enable	   := Para.bT_EGaLPTC_B_Active AND NOT Para.bT_EGaLPTC_HiTrip;
	xMsg2551.Set 	   := IN_EX.tPB2MM.bParaSetupOk AND NOT IN_EX.tT_EGaLPTC_B.GoodQual;
	xMsg2551.PT		   := T#0s;
	xMsg2551.Prio 	   := 4;
	xMsg2551.RiskClass := 4;
	xMsg2551.Reset     := FALSE;
	xMsg2551();
	MM2VIS.bMsg2551    := xMsg2551.Q;

	(* W2601 exhaust gas scavenging fan circuit breaker tripped *)
	xMsg2601.Enable	   := TRUE;
	xMsg2601.Set 	   := NOT IN_EX.tScavFanCB_trip.Di;
	xMsg2601.PT		   := T#0s;
	xMsg2601.Prio 	   := 4;
	xMsg2601.RiskClass := 4;
	xMsg2601.Reset     := FALSE;
	xMsg2601();
	MM2VIS.bMsg2601    := xMsg2601.Q;

	(* W2622 exhaust gas temperature high after low pressure turbo charger *)
	xMsg2622.Enable	   := TRUE;
	xMsg2622.Set 	   := FALSE;	(* 424tstc have to be specified *)
	xMsg2622.PT		   := T#0s;
	xMsg2622.Prio 	   := 4;
	xMsg2622.RiskClass := 4;
	xMsg2622.Reset     := FALSE;
	xMsg2622();
	MM2VIS.bMsg2622    := xMsg2622.Q;

	(* W2623 signal failure exhaust gas temperature after low pressure turbo charger *)
	xMsg2623.Enable	   := TRUE;
	xMsg2623.Set 	   := FALSE;	(* 424tstc have to be specified *)
	xMsg2623.PT		   := T#0s;
	xMsg2623.Prio 	   := 4;
	xMsg2623.RiskClass := 4;
	xMsg2623.Reset     := FALSE;
	xMsg2623();
	MM2VIS.bMsg2623    := xMsg2623.Q;

	(* W2655 signal failure exhaust gas temperature before high-pressure turbocharger A (M.02-TI-166)*)
	xMsg2655.Enable	   := Para.bT_EGbHPTC_A_Active;
	xMsg2655.Set 	   := IN_EX.tPB2MM.bParaSetupOk AND NOT IN_EX.tT_EGbHPTC_A.GoodQual;
	xMsg2655.PT		   := T#0s;
	xMsg2655.Prio 	   := 4;
	xMsg2655.RiskClass := 4;
	xMsg2655.Reset     := FALSE;
	xMsg2655();
	MM2VIS.bMsg2655    := xMsg2655.Q;

	(* W2656 signal failure exhaust gas temperature before high-pressure turbocharger B (M.02-TI-266)*)
	xMsg2656.Enable	   := Para.bT_EGbHPTC_B_Active;
	xMsg2656.Set 	   := IN_EX.tPB2MM.bParaSetupOk AND NOT IN_EX.tT_EGbHPTC_B.GoodQual;
	xMsg2656.PT		   := T#0s;
	xMsg2656.Prio 	   := 4;
	xMsg2656.RiskClass := 4;
	xMsg2656.Reset     := FALSE;
	xMsg2656();
	MM2VIS.bMsg2656    := xMsg2656.Q;

	(* W2657 signal failure exhaust gas temperatur after high-pressure turbocharger A (M.02-TI-167)*)
	xMsg2657.Enable	   := Para.bT_EGaHPTC_A_Active;
	xMsg2657.Set 	   := IN_EX.tPB2MM.bParaSetupOk AND NOT IN_EX.tT_EGaHPTC_A.GoodQual;
	xMsg2657.PT		   := T#0s;
	xMsg2657.Prio 	   := 4;
	xMsg2657.RiskClass := 4;
	xMsg2657.Reset     := FALSE;
	xMsg2657();
	MM2VIS.bMsg2657    := xMsg2657.Q;

	(* W2658 signal failure exhaust gas temperatur after high-pressure turbocharger B (M.02-TI-267)*)
	xMsg2658.Enable	   := Para.bT_EGaHPTC_B_Active;
	xMsg2658.Set 	   := IN_EX.tPB2MM.bParaSetupOk AND NOT IN_EX.tT_EGaHPTC_B.GoodQual;
	xMsg2658.PT		   := T#0s;
	xMsg2658.Prio 	   := 4;
	xMsg2658.RiskClass := 4;
	xMsg2658.Reset     := FALSE;
	xMsg2658();
	MM2VIS.bMsg2658    := xMsg2658.Q;

	(* W2659 signal failure exhaust gas pressure before high-pressure turbocharger A (M.02-PI-152)*)
	xMsg2659.Enable	   := Para.bPr_EGbHPTC_A_Active;
	xMsg2659.Set 	   := IN_EX.tPB2MM.bParaSetupOk AND NOT IN_EX.tPr_EGbHPTC_A.GoodQual;
	xMsg2659.PT		   := T#0s;
	xMsg2659.Prio 	   := 4;
	xMsg2659.RiskClass := 4;
	xMsg2659.Reset     := FALSE;
	xMsg2659();
	MM2VIS.bMsg2659    := xMsg2659.Q;

	(* W2660 exhaust gas pressure before high-pressure turbocharger B (M.02-PI-252)*)
	xMsg2660.Enable	   := Para.bPr_EGbHPTC_B_Active;
	xMsg2660.Set 	   := IN_EX.tPB2MM.bParaSetupOk AND NOT IN_EX.tPr_EGbHPTC_B.GoodQual;
	xMsg2660.PT		   := T#0s;
	xMsg2660.Prio 	   := 4;
	xMsg2660.RiskClass := 4;
	xMsg2660.Reset     := FALSE;
	xMsg2660();
	MM2VIS.bMsg2660    := xMsg2660.Q;

  	(* W2661 exhaust gas pressure after high-pressure turbocharger A (M.02-PI-153)*)
   	xMsg2661.Enable	   := Para.bPr_EGaHPTC_A_Active;
	xMsg2661.Set 	   := IN_EX.tPB2MM.bParaSetupOk AND NOT IN_EX.tPr_EGaHPTC_A.GoodQual;
	xMsg2661.PT		   := T#0s;
	xMsg2661.Prio 	   := 4;
	xMsg2661.RiskClass := 4;
	xMsg2661.Reset     := FALSE;
	xMsg2661();
	MM2VIS.bMsg2661    := xMsg2661.Q;

  	(* W2662 exhaust gas pressure after high-pressure turbocharger B (M.02-PI-253)*)
   	xMsg2662.Enable	   := Para.bPr_EGaHPTC_B_Active;
	xMsg2662.Set 	   := IN_EX.tPB2MM.bParaSetupOk AND NOT IN_EX.tPr_EGaHPTC_B.GoodQual;
	xMsg2662.PT		   := T#0s;
	xMsg2662.Prio 	   := 4;
	xMsg2662.RiskClass := 4;
	xMsg2662.Reset     := FALSE;
	xMsg2662();
	MM2VIS.bMsg2662    := xMsg2662.Q;

   	(* W2663 signal failure exhaust gas pressure after low-pressure turbocharger A (M.02-PI-154)*)
   	xMsg2663.Enable	   := Para.bPr_EGaLPTC_A_Active;
	xMsg2663.Set 	   := IN_EX.tPB2MM.bParaSetupOk AND NOT IN_EX.tPr_EGaLPTC_A.GoodQual;
	xMsg2663.PT		   := T#0s;
	xMsg2663.Prio 	   := 4;
	xMsg2663.RiskClass := 4;
	xMsg2663.Reset     := FALSE;
	xMsg2663();
	MM2VIS.bMsg2663    := xMsg2663.Q;

   	(* W2664 signal failure exhaust gas pressure after low-pressure turbocharger B (M.02-PI-254)*)
   	xMsg2664.Enable	   := Para.bPr_EGaLPTC_B_Active;
	xMsg2664.Set 	   := IN_EX.tPB2MM.bParaSetupOk AND NOT IN_EX.tPr_EGaLPTC_B.GoodQual;
	xMsg2664.PT		   := T#0s;
	xMsg2664.Prio 	   := 4;
	xMsg2664.RiskClass := 4;
	xMsg2664.Reset     := FALSE;
	xMsg2664();
	MM2VIS.bMsg2664    := xMsg2664.Q;

	(* W2743 meassuring signal failure differential pressure exhaust gas filter *)
	xMsg2743.Enable	   := Para.bPr_Diff_ExGFilter_Active;
	xMsg2743.Set 	   := NOT IN_EX.tPr_Diff_ExGFilter.GoodQual;
	xMsg2743.PT		   := T#0s;
	xMsg2743.Prio 	   := 4;
	xMsg2743.RiskClass := 4;
	xMsg2743.Reset     := FALSE;
	xMsg2743();
	MM2VIS.bMsg2743    := xMsg2743.Q;

	(* W2744 meassuring signal failure differential pressure exhaust gas cooler *)
	xMsg2744.Enable	   := Para.bPr_Diff_ExGCooler_Active;
	xMsg2744.Set 	   := NOT IN_EX.tPr_Diff_ExGCooler.GoodQual;
	xMsg2744.PT		   := T#0s;
	xMsg2744.Prio 	   := 4;
	xMsg2744.RiskClass := 4;
	xMsg2744.Reset     := FALSE;
	xMsg2744();
	MM2VIS.bMsg2744    := xMsg2744.Q;

	(* W2745 differential pressure exhaust gas ffilter maximum 1 *)
	xGR_MAXR_Pr_Diff_ExGFil_LimHi1(In:= IN_EX.tPr_Diff_ExGFilter.Ai, Gw:= Para.rPr_Diff_ExGFilter_Hi1, Hy:= Para.rPr_Diff_ExGFilter_HyHi);

	xMsg2745.Enable	   := Para.bPr_Diff_ExGFilter_Active;
	xMsg2745.Set 	   := xGR_MAXR_Pr_Diff_ExGFil_LimHi1.Q AND NOT MM2VIS.bMsg2743;
	xMsg2745.PT		   := T#2s;
	xMsg2745.Prio 	   := 4;
	xMsg2745.RiskClass := 4;
	xMsg2745.Reset     := FALSE;
	xMsg2745();
	MM2VIS.bMsg2745    := xMsg2745.Q;

	(* W2746 differential pressure exhaust gas ffilter maximum 2 *)
	xGR_MAXR_Pr_Diff_ExGFil_LimHi2(In:= IN_EX.tPr_Diff_ExGFilter.Ai, Gw:= Para.rPr_Diff_ExGFilter_Hi2, Hy:= Para.rPr_Diff_ExGFilter_HyHi);

	xMsg2746.Enable	   := Para.bPr_Diff_ExGFilter_Active;
	xMsg2746.Set 	   := xGR_MAXR_Pr_Diff_ExGFil_LimHi2.Q AND NOT MM2VIS.bMsg2743;
	xMsg2746.PT		   := T#2s;
	xMsg2746.Prio 	   := 4;
	xMsg2746.RiskClass := 4;
	xMsg2746.Reset     := FALSE;
	xMsg2746();
	MM2VIS.bMsg2746    := xMsg2746.Q;

	(* W2747 differential pressure exhaust gas ffilter minimum *)
	xGR_MINR_Pr_Diff_ExGFil_LimLo(In:= IN_EX.tPr_Diff_ExGFilter.Ai, Gw:= Para.rPr_Diff_ExGFilter_Lo, Hy:= Para.rPr_Diff_ExGFilter_HyHi);

	xMsg2747.Enable	   := Para.bPr_Diff_ExGFilter_Active;
	xMsg2747.Set 	   := xGR_MINR_Pr_Diff_ExGFil_LimLo.Q AND NOT MM2VIS.bMsg2743;
	xMsg2747.PT		   := T#2s;
	xMsg2747.Prio 	   := 4;
	xMsg2747.RiskClass := 4;
	xMsg2747.Reset     := FALSE;
	xMsg2747();
	MM2VIS.bMsg2747    := xMsg2747.Q;

	(* W2748 differential pressure exhaust gas coller maximum *)
	xGR_MAXR_Pr_Diff_ExGCoo_LimHi(In:= IN_EX.tPr_Diff_ExGCooler.Ai, Gw:= Para.rPr_Diff_ExGCooler_Hi, Hy:= Para.rPr_Diff_ExGCooler_HyHi);

	xMsg2748.Enable	   := Para.bPr_Diff_ExGCooler_Active;
	xMsg2748.Set 	   := xGR_MAXR_Pr_Diff_ExGCoo_LimHi.Q AND NOT MM2VIS.bMsg2744;
	xMsg2748.PT		   := T#2s;
	xMsg2748.Prio 	   := 4;
	xMsg2748.RiskClass := 4;
	xMsg2748.Reset     := FALSE;
	xMsg2748();
	MM2VIS.bMsg2748    := xMsg2748.Q;

	(* W2793 exhaust gas scavenging fan not ready *)
	xMsg2793.Enable	   := IN_EX.tPB2MM.bParaSetupOk;
	xMsg2793.Set 	   := NOT IN_EX.tScavFanFC_Rdy.Di;
	xMsg2793.PT		   := T#10s;
	xMsg2793.Prio 	   := 4;
	xMsg2793.RiskClass := 4;
	xMsg2793.Reset     := FALSE;
	xMsg2793();
	MM2VIS.bMsg2793    := xMsg2793.Q;

	(* A3100 exhaust gas temperature before turbo charger high *)
	xGR_MAXR_T_EGbTC_LimHiHi(In:= IN_EX.tT_EGbTC.Ai, Gw:= Para.rT_EGbTC_LimHiHi, Hy:= Para.rT_EGbTC_HyHiHi);

//	xMsg3100.Enable	   := Para.bT_EGbTC_Active AND NOT xEngType.Type9;//SWAT920/2 --> ELIMINATE SWAT MODIFICATION BACK TO OLD VERSION! 09.10.2017 TW
	xMsg3100.Enable	   := Para.bT_EGbTC_Active;
	xMsg3100.Set 	   := xGR_MAXR_T_EGbTC_LimHiHi.Q AND IN_EX.tPB2MM.bParaSetupOk AND NOT MM2VIS.bMsg3214;
//	xMsg3100.PT		   := T#2s;
	xMsg3100.PT		   := T#122s;	//SWAT920/x increase time delay from 2s to 120s! 09.10.2017 TW
	xMsg3100.Prio 	   := 3;
	xMsg3100.RiskClass := 4;
	xMsg3100.Reset     := FALSE;
	xMsg3100();
	MM2VIS.bMsg3100    := xMsg3100.Q;

	(* W3214 exhaust gas temperature before turbo charger signal failure *)
	xMsg3214.Enable	   := Para.bT_EGbTC_Active;
	xMsg3214.Set 	   := IN_EX.tPB2MM.bParaSetupOk AND NOT IN_EX.tT_EGbTC.GoodQual;
	xMsg3214.PT		   := T#0s;
	xMsg3214.Prio 	   := 4;
	xMsg3214.RiskClass := 4;
	xMsg3214.Reset     := FALSE;
	xMsg3214();
	MM2VIS.bMsg3214	   := xMsg3214.Q;

	(* W3215 exhaust gas temperature before turbo charger high *)
	xGR_MAXR_T_EGbTC_LimHi(In:= IN_EX.tT_EGbTC.Ai, Gw:= Para.rT_EGbTC_LimHi, Hy:= Para.rT_EGbTC_HyHi);

	xMsg3215.Enable	   := Para.bT_EGbTC_Active;
	xMsg3215.Set 	   := xGR_MAXR_T_EGbTC_LimHi.Q AND IN_EX.tPB2MM.bParaSetupOk AND NOT MM2VIS.bMsg3214;
	xMsg3215.PT		   := T#2s;
	xMsg3215.Prio 	   := 4;
	xMsg3215.RiskClass := 4;
	xMsg3215.Reset     := FALSE;
	xMsg3215();
	MM2VIS.bMsg3215    := xMsg3215.Q;

	(* A3313 CODINOX: CO2 reactor chamber temperature high *)
	xMsg3313.Enable	   := Para.bCodinox_Active;
	xMsg3313.Set 	   := IN_EX.tT_CO2_Hi.Di;
	xMsg3313.PT		   := T#0s;
	xMsg3313.Prio 	   := 2;
	xMsg3313.RiskClass := 4;
	xMsg3313.Reset     := FALSE;
	xMsg3313();
	MM2VIS.bMsg3313    := xMsg3313.Q;

   (* A3314 CODINOX: CO2 valve failure *)
    xMsg3314.Enable	   := Para.bCodinox_Active;
	xMsg3314.Set 	   := CO2KLST_A;
	xMsg3314.PT		   := T#0s;
	xMsg3314.Prio 	   := 2;
	xMsg3314.RiskClass := 4;
	xMsg3314.Reset     := FALSE;
	xMsg3314();
	MM2VIS.bMsg3314    := xMsg3314.Q;

    (* W3349 N2 gas valves position failure *)
    xMsg3349.Enable	   := Para.bSel_N2;
	xMsg3349.Set 	   := (bOMSS_MAT OR bOMSS_Scav) AND T1_STN2V;
	xMsg3349.PT		   := T#0s;
	xMsg3349.Prio 	   := 2;
	xMsg3349.RiskClass := 4;
	xMsg3349.Reset     := FALSE;
	xMsg3349();
	MM2VIS.bMsg3349    := xMsg3349.Q;

	(********************************************************************************************************************
	Safety-related application software source code (EN 13849-1 / 4.6.3): BEGIN
	*********************************************************************************************************************)

	(* A3366 exhaust gas scavenging fan failure (W1165) *)
	xMsg3366.Enable	   := NOT xEngType.Type9;//SWAT920/5
	xMsg3366.Set 	   :=	OUT_EX.tScavFanCoOn.Do AND NOT IN_EX.tEng_Run.Do
					AND NOT bNoMon4BlackStart
				AND(	(NOT xEngType.Type9 AND NOT IN_EX.tScavFanOp.Di AND NOT NoScavFan)
					OR	(    xEngType.Type9 AND    (IN_EX.tScavFanFC_P_Lo.Di OR NOT IN_EX.tScavFanFC_Rdy.Di)));
	xMsg3366.PT		   := T#10s;
	xMsg3366.Prio 	   := 3;
	xMsg3366.RiskClass := 10;
	xMsg3366.Reset     := FALSE;
	xMsg3366();
	MM2VIS.bMsg3366	   := xMsg3366.Q;

	(********************************************************************************************************************
	Safety-related application software source code (EN 13849-1 / 4.6.3): END
	*********************************************************************************************************************)

	(* A3394 exhaust gas temperature after exhaust heat exchanger 1 high *) (*STM*)
	xGR_MAXR_T_EGaHE1_LimHi_Trip(In:= IN_EX.tT_EGaHE1.Ai, Gw:= Para.rT_EGaHE1_LimHi_Trip, Hy:= Para.rT_EGaHE1_HyHi_Trip);
	bT_EGaHE1_LimHi_Trip := xGR_MAXR_T_EGaHE1_LimHi_Trip.Q;

	xMsg3394.Enable	   := Para.bT_EGaHE1_Active;
	xMsg3394.Set 	   := bT_EGaHE1_LimHi_Trip AND NOT MM2VIS.bMsg3513;
	xMsg3394.PT		   := T#2s;
	xMsg3394.Prio 	   := 3;
	xMsg3394.RiskClass := 4;
	xMsg3394.Reset     := FALSE;
	xMsg3394();
	MM2VIS.bMsg3394    := xMsg3394.Q;

	(* A3395 exhaust gas temperature after exhaust heat exchanger 2 high *) (*STM*)
	xGR_MAXR_T_EGaHE2_LimHi_Trip(In:= IN_EX.tT_EGaHE2.Ai, Gw:= Para.rT_EGaHE2_LimHi_Trip, Hy:= Para.rT_EGaHE2_HyHi_Trip);
	bT_EGaHE2_LimHi_Trip := xGR_MAXR_T_EGaHE2_LimHi_Trip.Q;

	xMsg3395.Enable	   := Para.bT_EGaHE2_Active;
	xMsg3395.Set 	   := bT_EGaHE2_LimHi_Trip AND NOT MM2VIS.bMsg3514;
	xMsg3395.PT		   := T#2s;
	xMsg3395.Prio 	   := 3;
	xMsg3395.RiskClass := 4;
	xMsg3395.Reset     := FALSE;
	xMsg3395();
	MM2VIS.bMsg3395    := xMsg3395.Q;

	(* A3397 differential pressure exhaust gas filter maximum *)
	xGR_MAXR_Pr_Diff_ExGFil_LimHiA(In:= IN_EX.tPr_Diff_ExGFilter.Ai, Gw:= Para.rPr_Diff_ExGFilter_Hi, Hy:= Para.rPr_Diff_ExGFilter_HyHi);

	xMsg3397.Enable	   := Para.bPr_Diff_ExGFilter_Active;
	xMsg3397.Set 	   := xGR_MAXR_Pr_Diff_ExGFil_LimHiA.Q AND NOT MM2VIS.bMsg2743;
	xMsg3397.PT		   := T#0s;
	xMsg3397.Prio 	   := 3;
	xMsg3397.RiskClass := 4;
	xMsg3397.Reset     := FALSE;
	xMsg3397();
	MM2VIS.bMsg3397    := xMsg3397.Q;

	(* W3417 pre chamber diff.pressure high during  engine stop (exhaust gas scavenging required before next start) *)
	xTON_Pr_PC_Diff_MonRel(IN:= StopM, PT:= T#30s);
	rPr_PC_Diff := IN_EX.tPr_PC.Ai - MAX(IN_EX.tPr_Ch_P2s.Ai, MAX(IN_EX.tPr_Ch_P2s_A.Ai, IN_EX.tPr_Ch_P2s_B.Ai)); (* calc.pre chamber diff.pressure *)

	xMsg3417.Enable	   := (Para.bEGScav_Active OR Para.bSel_N2 OR xEngType.Type6)
				   AND NOT xEngType.Type9;
	xMsg3417.Set 	   := (rPr_PC_Diff > Para.rPr_PC_Diff_LimHi) AND xTON_Pr_PC_Diff_MonRel.Q AND NOT IN_EX.bMsg1078;
	xMsg3417.PT		   := T#5s;
	xMsg3417.Prio 	   := 4;
	xMsg3417.RiskClass := 4;
	xMsg3417.Reset     := FALSE;
	xMsg3417();
	MM2VIS.bMsg3417	   := xMsg3417.Q;

	(* W3490 exhaust gas temperature after exhaust heat exchanger 1 high *) (*STM*)
	xGR_MAXR_T_EGaHE1_LimHi_Warn(In:= IN_EX.tT_EGaHE1.Ai, Gw:= Para.rT_EGaHE1_LimHi_Warn, Hy:= Para.rT_EGaHE1_HyHi_Warn);
	bT_EGaHE1_LimHi_Warn := xGR_MAXR_T_EGaHE1_LimHi_Warn.Q;

	xMsg3490.Enable	   := Para.bT_EGaHE1_Active;
	xMsg3490.Set 	   := bT_EGaHE1_LimHi_Warn AND NOT MM2VIS.bMsg3513;
	xMsg3490.PT		   := T#2s;
	xMsg3490.Prio 	   := 4;
	xMsg3490.RiskClass := 4;
	xMsg3490.Reset     := FALSE;
	xMsg3490();
	MM2VIS.bMsg3490    := xMsg3490.Q;

	(* W3491 exhaust gas temperature after exhaust heat exchanger 2 high *) (*STM*)
	xGR_MAXR_T_EGaHE2_LimHi_Warn(In:= IN_EX.tT_EGaHE2.Ai, Gw:= Para.rT_EGaHE2_LimHi_Warn, Hy:= Para.rT_EGaHE2_HyHi_Warn);
	bT_EGaHE2_LimHi_Warn := xGR_MAXR_T_EGaHE2_LimHi_Warn.Q;

	xMsg3491.Enable	   := Para.bT_EGaHE2_Active;
	xMsg3491.Set 	   := bT_EGaHE2_LimHi_Warn AND NOT MM2VIS.bMsg3514;
	xMsg3491.PT		   := T#2s;
	xMsg3491.Prio 	   := 4;
	xMsg3491.RiskClass := 4;
	xMsg3491.Reset     := FALSE;
	xMsg3491();
	MM2VIS.bMsg3491    := xMsg3491.Q;

	(* W3510 CODINOX: CO2 Ventilation fan failure *)
	xMsg3510.Enable	   := Para.bCodinox_Active;
	xMsg3510.Set 	   := NOT IN_EX.tCO2_FanFailure.Di;
	xMsg3510.PT		   := T#0s;
	xMsg3510.Prio 	   := 4;
	xMsg3510.RiskClass := 4;
	xMsg3510.Reset     := TRUE;	(* autoreset customers request *)
	xMsg3510();
	MM2VIS.bMsg3510    := xMsg3510.Q;

	(* W3511 CODINOX: CO2 station failure *)
	xMsg3511.Enable	   := Para.bCodinox_Active;
	xMsg3511.Set 	   := NOT IN_EX.tCO2_DevFailure.Di;
	xMsg3511.PT		   := T#0s;
	xMsg3511.Prio 	   := 4;
	xMsg3511.RiskClass := 4;
	xMsg3511.Reset     := TRUE;	(* autoreset customers request *)
	xMsg3511();
	MM2VIS.bMsg3511    := xMsg3511.Q;

	(* W3512 CODINOX: CO2 valve failure *)
	xMsg3512.Enable	   := Para.bCodinox_Active;
	xMsg3512.Set 	   := CO2KLST_W;
	xMsg3512.PT		   := T#0s;
	xMsg3512.Prio 	   := 4;
	xMsg3512.RiskClass := 4;
	xMsg3512.Reset     := FALSE;
	xMsg3512();
	MM2VIS.bMsg3512    := xMsg3512.Q;

	(* W3513 CODINOX: exhaust gas temperature after heat exchanger 1 measuring signal failure *)
	xMsg3513.Enable	   := Para.bT_EGaHE1_Active;
	xMsg3513.Set 	   := IN_EX.tPB2MM.bParaSetupOk AND NOT IN_EX.tT_EGaHE1.GoodQual;
	xMsg3513.PT		   := T#0s;
	xMsg3513.Prio 	   := 4;
	xMsg3513.RiskClass := 4;
	xMsg3513.Reset     := FALSE;
	xMsg3513();
	MM2VIS.bMsg3513    := xMsg3513.Q;

	(* W3514 CODINOX: exhaust gas temperature after heat exchanger 2 measuring signal failure *)
	xMsg3514.Enable	   := Para.bT_EGaHE2_Active;
	xMsg3514.Set 	   := IN_EX.tPB2MM.bParaSetupOk AND NOT IN_EX.tT_EGaHE2.GoodQual;
	xMsg3514.PT		   := T#0s;
	xMsg3514.Prio 	   := 4;
	xMsg3514.RiskClass := 4;
	xMsg3514.Reset     := FALSE;
	xMsg3514();
	MM2VIS.bMsg3514    := xMsg3514.Q;

	(********************************************************************************************************************
	Safety-related application software source code (EN 13849-1 / 4.6.3): BEGIN
	*********************************************************************************************************************)

	(* W3528 exhaust gas back pressure high *)
	xMsg3528.Enable	   := NOT Para.bSafe_Pr_EG_sMonActive; 						(* SAFETY PLC *)
	xMsg3528.Set 	   := NOT IN_EX.tPr_EG_Hi.Di;
	xMsg3528.PT		   := T#5s;
	xMsg3528.Prio 	   := 4;
	xMsg3528.RiskClass := 4;
	xMsg3528.Reset     := FALSE;
	xMsg3528();
	MM2VIS.bMsg3528    := xMsg3528.Q;

	(********************************************************************************************************************
	Safety-related application software source code (EN 13849-1 / 4.6.3): END
	*********************************************************************************************************************)

	(* W3580 N2 gas pressure low *)
	xMsg3580.Enable	   := Para.bSel_N2;
	xMsg3580.Set 	   := (bOMSS_MAT OR bOMSS_Scav) AND OUT_EX.bPr_N2_LoTon;
	xMsg3580.PT		   := T#0s;
	xMsg3580.Prio 	   := 4;
	xMsg3580.RiskClass := 4;
	xMsg3580.Reset     := FALSE;
	xMsg3580();
	MM2VIS.bMsg3580    := xMsg3580.Q;

	(* W3581 N2 gas pressure high *)
	xMsg3581.Enable	   := Para.bSel_N2;
	xMsg3581.Set 	   := (bOMSS_MAT OR bOMSS_Scav) AND NOT IN_EX.tPr_N2_Hi.Di;
	xMsg3581.PT		   := T#5s;
	xMsg3581.Prio 	   := 4;
	xMsg3581.RiskClass := 4;
	xMsg3581.Reset     := FALSE;
	xMsg3581();
	MM2VIS.bMsg3581    := xMsg3581.Q;

	(* W3582 N2 scavenging run failure *)
	xMsg3582.Enable	   := Para.bSel_N2;
	xMsg3582.Set 	   := (bOMSS_MAT OR bOMSS_Scav) AND (T1_SCAV_RUN OR T2_SCAV_RUN);
	xMsg3582.PT		   := T#0s;
	xMsg3582.Prio 	   := 4;
	xMsg3582.RiskClass := 4;
	xMsg3582.Reset     := FALSE;
	xMsg3582();
	MM2VIS.bMsg3582    := xMsg3582.Q;

	(* W9215 air temperature before exhaust gas scavening valve maximum *)//SWAT920/5
	xMsg9215.Enable	   := Para.bT_bScavValve_Active;
	xMsg9215.Set 	   := IN_EX.tPB2MM.bParaSetupOk AND  IN_EX.tT_bScavValve.GoodQual
													AND (IN_EX.tT_bScavValve.Ai > Para.rT_bScavValve_LimHi1);
	xMsg9215.PT		   := T#2s;
	xMsg9215.Prio 	   := 4;
	xMsg9215.RiskClass := 4;
	xMsg9215.Reset     := FALSE;
	xMsg9215();
	MM2VIS.bMsg9215    := xMsg9215.Q;

	(* W9249 Exhaust gas pressure fast measurement signal failure (W2497) *)	//blocks engine restart if active

	xMsg9249.Enable	   := Para.bPr_OXIcat_In_Fast_Exist;
	xMsg9249.Set 	   := NOT IN_EX.tPr_EG_Deflag_Fast.GoodQual;
	xMsg9249.PT		   := T#0s;
	xMsg9249.Prio 	   := 4;
	xMsg9249.RiskClass := 4;
	xMsg9249.Reset     := FALSE;
	xMsg9249();
	MM2VIS.bMsg9249    := xMsg9249.Q;
	OUT_EX.bMsg9249    := xMsg9249.Q;

	(* W9305 (A2337) temperature high exhaust gas pressure relief valve 1 *)(* P.02-TI-039 *)
	xMsg9305.Enable	   := Para.bT_EG_PrReliefVa1_Active;
	xMsg9305.Set 	   := IN_EX.tPB2MM.bParaSetupOk AND(IN_EX.tT_EG_PrReliefVa1.Ai > Para.rT_EG_PrReliefVa_LimHi) AND NOT MM2VIS.bMsg9307;
	xMsg9305.PT		   := T#2s;
	xMsg9305.Prio 	   := 4;
	xMsg9305.RiskClass := 4;
	xMsg9305.Reset     := FALSE;
	xMsg9305();
	MM2VIS.bMsg9305    := xMsg9305.Q;

	(* W9306 (A2338) temperature high exhaust gas pressure relief valve 2 *)(* P.02-TI-040 *)
	xMsg9306.Enable	   := Para.bT_EG_PrReliefVa2_Active;
	xMsg9306.Set 	   := IN_EX.tPB2MM.bParaSetupOk AND(IN_EX.tT_EG_PrReliefVa2.Ai > Para.rT_EG_PrReliefVa_LimHi) AND NOT MM2VIS.bMsg9308;
	xMsg9306.PT		   := T#2s;
	xMsg9306.Prio 	   := 4;
	xMsg9306.RiskClass := 4;
	xMsg9306.Reset     := FALSE;
	xMsg9306();
	MM2VIS.bMsg9306    := xMsg9306.Q;

	(* W9307 temperature exhaust gas pressure relief valve 1 signal failure *)(* P.02-TI-039 *)
	xMsg9307.Enable	   := Para.bT_EG_PrReliefVa1_Active;
	xMsg9307.Set 	   := IN_EX.tPB2MM.bParaSetupOk AND NOT IN_EX.tT_EG_PrReliefVa1.GoodQual;
	xMsg9307.PT		   := T#0s;
	xMsg9307.Prio 	   := 4;
	xMsg9307.RiskClass := 4;
	xMsg9307.Reset     := FALSE;
	xMsg9307();
	MM2VIS.bMsg9307    := xMsg9307.Q;

	(* W9308 temperature exhaust gas pressure relief valve 2 signal failure *)(* P.02-TI-040 *)
	xMsg9308.Enable	   := Para.bT_EG_PrReliefVa2_Active;
	xMsg9308.Set 	   := IN_EX.tPB2MM.bParaSetupOk AND NOT IN_EX.tT_EG_PrReliefVa2.GoodQual;
	xMsg9308.PT		   := T#0s;
	xMsg9308.Prio 	   := 4;
	xMsg9308.RiskClass := 4;
	xMsg9308.Reset     := FALSE;
	xMsg9308();
	MM2VIS.bMsg9308    := xMsg9308.Q;

	(* W9310 OXIcat Outlet temperature measurement signal failure *)(* A2319 *)
	xMsg9310.Enable	   := Para.bOXIcat_Exist
					  AND Para.bT_OXIcat_Out_Exist;
	xMsg9310.Set 	   := NOT IN_EX.tT_EGaCat.GoodQual
					  AND (IN_EX.rN_EngAct > 0);
	xMsg9310.PT		   := T#60s;
	xMsg9310.Prio 	   := 4;
	xMsg9310.RiskClass := 4;
	xMsg9310.Reset     := FALSE;
	xMsg9310();
	MM2VIS.bMsg9310    := xMsg9310.Q;

	(* W9347 exhaust gas flaps - module standstill position not reached *)
	(*                          = bypass open, boiler closed *)
	xTON_9347(IN:= NOT IN_EX.tEng_Run.Do AND ((NOT IN_EX.tEG_ByVaOpened.Di AND IN_EX.tEG_ByVaOpened.GoodQual)
					  					  OR  (NOT IN_EX.tEG_BoVaClosed.Di AND IN_EX.tEG_BoVaClosed.GoodQual)), PT:= T#60s);

	xMsg9347.Enable	   := IN_EX.tPB2MM.bSys_Run;
	xMsg9347.Set 	   := xTON_9347.Q;
	xMsg9347.PT		   := T#0s;
	xMsg9347.Prio 	   := 4;
	xMsg9347.RiskClass := 4;
	xMsg9347.Reset     := FALSE;
	xMsg9347();
	MM2VIS.bMsg9347    := xMsg9347.Q;

	OUT_EX.bEngBloc_EX := xMsg9347.Set;

	(* W9348 exhaust gas flaps - status signal failure *)
	xMsg9348.Enable	   := IN_EX.tPB2MM.bSys_Run;
	xMsg9348.Set 	   := (    IN_EX.tEG_ByVaOpened.Di AND     IN_EX.tEG_ByVaClosed.Di AND IN_EX.tEG_ByVaOpened.GoodQual AND IN_EX.tEG_ByVaClosed.GoodQual)
					   OR (NOT IN_EX.tEG_ByVaOpened.Di AND NOT IN_EX.tEG_ByVaClosed.Di AND IN_EX.tEG_ByVaOpened.GoodQual AND IN_EX.tEG_ByVaClosed.GoodQual)
					   OR (    IN_EX.tEG_BoVaOpened.Di AND     IN_EX.tEG_BoVaClosed.Di AND IN_EX.tEG_BoVaOpened.GoodQual AND IN_EX.tEG_BoVaClosed.GoodQual)
					   OR (NOT IN_EX.tEG_BoVaOpened.Di AND NOT IN_EX.tEG_BoVaClosed.Di AND IN_EX.tEG_BoVaOpened.GoodQual AND IN_EX.tEG_BoVaClosed.GoodQual);
	xMsg9348.PT		   := T#60s;
	xMsg9348.Prio 	   := 4;
	xMsg9348.RiskClass := 4;
	xMsg9348.Reset     := FALSE;
	xMsg9348();
	MM2VIS.bMsg9348    := xMsg9348.Q;

	(*---------------------------------------------------------------------------*)
	(* operating messages > AMM *)

	(* B1273 demand exhaust gas scavenging flap open *)
	xMsg1273.Enable		:=	xEngType.Type9 OR Para.bEGScav_Active;
	xMsg1273.Set		:=	OUT_EX.tScavVaCoOpen.Do;
	xMsg1273.Reset		:=	TRUE;
	xMsg1273();
	MM2VIS.bMsg1273		:=	xMsg1273.Q;

	(* B1274 demand exhaust gas scavenging flap close *)
	xMsg1274.Enable		:=	xEngType.Type9 OR Para.bEGScav_Active;
	xMsg1274.Set		:=	OUT_EX.tScavVaCoClose.Do AND IN_EX.tPB2MM.bSys_Run;
	xMsg1274.Reset		:=	TRUE;
	xMsg1274();
	MM2VIS.bMsg1274		:=	xMsg1274.Q;

	(* B1275 exhaust gas scavenging valve opened *)
	xMsg1275.Enable		:=	xEngType.Type9 OR Para.bEGScav_Active;
	xMsg1275.Set		:=	IN_EX.tScavVaOpened.Di AND NOT IN_EX.tScavVaClosed.Di;
	xMsg1275.Reset		:=	TRUE;
	xMsg1275();
	MM2VIS.bMsg1275		:=	xMsg1275.Q;

	(* B1276 exhaust gas scavenging valve closed *)
	xMsg1276.Enable		:=	xEngType.Type9 OR Para.bEGScav_Active;
	xMsg1276.Set		:=	IN_EX.tScavVaClosed.Di AND NOT IN_EX.tScavVaOpened.Di AND IN_EX.tPB2MM.bSys_Run;
	xMsg1276.Reset		:=	TRUE;
	xMsg1276();
	MM2VIS.bMsg1276		:=	xMsg1276.Q;

	(* B1277 demand exhaust gas scavenging fan on *)
	xMsg1277.Enable		:=	xEngType.Type9 OR Para.bEGScav_Active;
	xMsg1277.Set		:=	    OUT_EX.tScavFanCoOn.Do AND IN_EX.tPB2MM.bSys_Run;
	xMsg1277.Reset		:=	TRUE;
	xMsg1277();
	MM2VIS.bMsg1277		:=	xMsg1277.Q;

	(* B1278 demand exhaust gas scavenging fan off *)
	xMsg1278.Enable		:=	xEngType.Type9 OR Para.bEGScav_Active;
	xMsg1278.Set		:=	NOT OUT_EX.tScavFanCoOn.Do AND IN_EX.tPB2MM.bSys_Run;
	xMsg1278.Reset		:=	TRUE;
	xMsg1278();
	MM2VIS.bMsg1278		:=	xMsg1278.Q;

	(* B1279 exhaust gas scavenging fan operation on *)
	xMsg1279.Enable		:=	xEngType.Type9 OR Para.bEGScav_Active;
	IF xEngType.Type9 THEN xMsg1279.Set := IN_EX.tScavFanFC_Rdy.Di AND NOT IN_EX.tScavFanFC_P_Lo.Di AND OUT_EX.tScavFanCoOn.Do;
	ELSE				   xMsg1279.Set := IN_EX.tScavFanOp.Di AND NOT NoScavFan;
	END_IF;
	xMsg1279.Reset		:=	TRUE;
	xMsg1279();
	MM2VIS.bMsg1279		:=	xMsg1279.Q;

	(* B1280 exhaust gas scavenging fan operation off *)
	xMsg1280.Enable		:=	xEngType.Type9 OR Para.bEGScav_Active;
	IF xEngType.Type9 THEN xMsg1280.Set := IN_EX.tPB2MM.bSys_Run AND NOT xMsg1279.Set;
	ELSE				   xMsg1280.Set := IN_EX.tPB2MM.bSys_Run AND NOT IN_EX.tScavFanOp.Di AND NOT NoScavFan;
	END_IF;
	xMsg1280.Reset		:=	TRUE;
	xMsg1280();
	MM2VIS.bMsg1280		:=	xMsg1280.Q;

	(* B1288 CO2 flap open *)
	xMsg1288.Enable		:=	Para.bCodinox_Active;
	xMsg1288.Set		:=	IN_EX.tCO2_VaOpened.Di;
	xMsg1288.Reset		:=	TRUE;
	xMsg1288();
	MM2VIS.bMsg1288		:=	xMsg1288.Q;

	(* B1289 CO2 flap closed *)
	xMsg1289.Enable		:=	Para.bCodinox_Active;
	xMsg1289.Set		:=	IN_EX.tCO2_VaClosed.Di;
	xMsg1289.Reset		:=	TRUE;
	xMsg1289();
	MM2VIS.bMsg1289		:=	xMsg1289.Q;

	(* B1290 CO2 demand on *)
	xMsg1290.Enable		:=	Para.bCodinox_Active;
	xMsg1290.Set		:=	IN_EX.tCO2_Demand.Di;
	xMsg1290.Reset		:=	TRUE;
	xMsg1290();
	MM2VIS.bMsg1290		:=	xMsg1290.Q;

	(* B1291 CO2 demand off *)
	xMsg1291.Enable		:=	Para.bCodinox_Active;
	xMsg1291.Set		:=	NOT IN_EX.tCO2_Demand.Di;
	xMsg1291.Reset		:=	TRUE;
	xMsg1291();
	MM2VIS.bMsg1291:=	xMsg1291.Q;

	(* 2847 N2 gas valves closed *)
	xMsg2847.Enable	   := Para.bSel_N2;
	xMsg2847.Set 	   := NOT OUT_EX.tN2_ScavGV_CoOpen.Do;
	xMsg2847.Reset     := TRUE;
	xMsg2847();
	MM2VIS.bMsg2847    := xMsg2847.Q;

	(* 2848 N2 gas valves opened *)
	xMsg2848.Enable	   := Para.bSel_N2;
	xMsg2848.Set 	   :=     OUT_EX.tN2_ScavGV_CoOpen.Do;
	xMsg2848.Reset     := TRUE;
	xMsg2848();
	MM2VIS.bMsg2848    := xMsg2848.Q;

	(* B template
	xMsg.Enable		:=	TRUE;
	xMsg.Set		:=	bBool;
	xMsg.Reset		:=	TRUE;
	xMsg();
	MM2VIS.bMsg		:=	xMsg.Q;	*)

	(*---------------------------------------------------------------------------*)
	(* general alarms for further module operations *)
	bGnlTrip1   := OUT_EX.tEX2AB.bGnlTrip1   OR IN_EX.tAB2EX.bGnlTrip1;
	bGnlTrip2   := OUT_EX.tEX2AB.bGnlTrip2   OR IN_EX.tAB2EX.bGnlTrip2;
	bGnlTrip3   := OUT_EX.tEX2AB.bGnlTrip3   OR IN_EX.tAB2EX.bGnlTrip3;
	bGnlWarning := OUT_EX.tEX2AB.bGnlWarning OR IN_EX.tAB2EX.bGnlWarning;

	bGnlTrip	:= bGnlTrip1 OR bGnlTrip2 OR bGnlTrip3;

	(*******************************************************************************)
END_PROGRAM
```

#### MsgEXInit.st
```iecst
(*******************************************************************************
Msg_EX	 			 alarms generation

This code is confidential and proprietary to the INNIO Company.
It may not be used in any form, or reproduced in any manner,
without written permission of the INNIO Company.
Copyright, INNIO Company, 2019

Customized modifications: -
------------------------

History:
-------
V0.00.0	29.07.2011	lettenb.	new
V4.13.0	19.10.2023	Heim Markus	add 2374

Instructions for use:
--------------------
1) declare alarm with function block "Msg"

2) use template to create a new alarm, substitue 0000 by message number:

	xMsg0000.Num		:=	0000;					alarm number
	xMsg0000.AmmSysAdr	:=  iAdrAmmBase2MM;			do not change
	xMsg0000.AmmOutAdr	:=  iAdrMM2AmmBase;			do not change

3) 	set alarm number

Outstandings:
------------
(*******************************************************************************)
PROGRAM _INIT

	iAdrAmmBase2MM		:=  ADR(IN_EX.tAB2EX);
	iAdrMM2AmmBase		:=  ADR(OUT_EX.tEX2AB);
	(*---------------------------------------------------------------------------*)

	xMsg1045.Num		:=	1045;
	xMsg1045.AmmInAdr	:=  iAdrAmmBase2MM;
	xMsg1045.AmmOutAdr	:=  iAdrMM2AmmBase;

	xMsg1046.Num		:=	1046;
	xMsg1046.AmmInAdr	:=  iAdrAmmBase2MM;
	xMsg1046.AmmOutAdr	:=  iAdrMM2AmmBase;

	xMsg1069.Num		:=	1069;
	xMsg1069.AmmInAdr	:=  iAdrAmmBase2MM;
	xMsg1069.AmmOutAdr	:=  iAdrMM2AmmBase;

	xMsg1092.Num		:=	1092;
	xMsg1092.AmmInAdr	:=  iAdrAmmBase2MM;
	xMsg1092.AmmOutAdr	:=  iAdrMM2AmmBase;

	xMsg1104.Num		:=	1104;
	xMsg1104.AmmInAdr	:=  iAdrAmmBase2MM;
	xMsg1104.AmmOutAdr	:=  iAdrMM2AmmBase;

	xMsg1106.Num		:=	1106;
	xMsg1106.AmmInAdr	:=  iAdrAmmBase2MM;
	xMsg1106.AmmOutAdr	:=  iAdrMM2AmmBase;

	xMsg1161.Num		:=	1161;
	xMsg1161.AmmInAdr	:=  iAdrAmmBase2MM;
	xMsg1161.AmmOutAdr	:=  iAdrMM2AmmBase;

	xMsg1162.Num		:=	1162;
	xMsg1162.AmmInAdr	:=  iAdrAmmBase2MM;
	xMsg1162.AmmOutAdr	:=  iAdrMM2AmmBase;

	xMsg1163.Num		:=	1163;
	xMsg1163.AmmInAdr	:=  iAdrAmmBase2MM;
	xMsg1163.AmmOutAdr	:=  iAdrMM2AmmBase;

	xMsg1164.Num		:=	1164;
	xMsg1164.AmmInAdr	:=  iAdrAmmBase2MM;
	xMsg1164.AmmOutAdr	:=  iAdrMM2AmmBase;

	xMsg1165.Num		:=	1165;
	xMsg1165.AmmInAdr	:=  iAdrAmmBase2MM;
	xMsg1165.AmmOutAdr	:=  iAdrMM2AmmBase;

	xMsg1169.Num		:=	1169;
	xMsg1169.AmmInAdr	:=  iAdrAmmBase2MM;
	xMsg1169.AmmOutAdr	:=  iAdrMM2AmmBase;

	xMsg1170.Num		:=	1170;
	xMsg1170.AmmInAdr	:=  iAdrAmmBase2MM;
	xMsg1170.AmmOutAdr	:=  iAdrMM2AmmBase;

	xMsg1171.Num		:=	1171;
	xMsg1171.AmmInAdr	:=  iAdrAmmBase2MM;
	xMsg1171.AmmOutAdr	:=  iAdrMM2AmmBase;

	xMsg1172.Num		:=	1172;
	xMsg1172.AmmInAdr	:=  iAdrAmmBase2MM;
	xMsg1172.AmmOutAdr	:=  iAdrMM2AmmBase;

	xMsg1173.Num		:=	1173;
	xMsg1173.AmmInAdr	:=  iAdrAmmBase2MM;
	xMsg1173.AmmOutAdr	:=  iAdrMM2AmmBase;

	xMsg1174.Num		:=	1174;
	xMsg1174.AmmInAdr	:=  iAdrAmmBase2MM;
	xMsg1174.AmmOutAdr	:=  iAdrMM2AmmBase;

	xMsg1273.Num		:=	1273;
	xMsg1273.AmmInAdr	:=  iAdrAmmBase2MM;
	xMsg1273.AmmOutAdr	:=  iAdrMM2AmmBase;

	xMsg1274.Num		:=	1274;
	xMsg1274.AmmInAdr	:=  iAdrAmmBase2MM;
	xMsg1274.AmmOutAdr	:=  iAdrMM2AmmBase;

	xMsg1275.Num		:=	1275;
	xMsg1275.AmmInAdr	:=  iAdrAmmBase2MM;
	xMsg1275.AmmOutAdr	:=  iAdrMM2AmmBase;

	xMsg1276.Num		:=	1276;
	xMsg1276.AmmInAdr	:=  iAdrAmmBase2MM;
	xMsg1276.AmmOutAdr	:=  iAdrMM2AmmBase;

	xMsg1277.Num		:=	1277;
	xMsg1277.AmmInAdr	:=  iAdrAmmBase2MM;
	xMsg1277.AmmOutAdr	:=  iAdrMM2AmmBase;

	xMsg1278.Num		:=	1278;
	xMsg1278.AmmInAdr	:=  iAdrAmmBase2MM;
	xMsg1278.AmmOutAdr	:=  iAdrMM2AmmBase;

	xMsg1279.Num		:=	1279;
	xMsg1279.AmmInAdr	:=  iAdrAmmBase2MM;
	xMsg1279.AmmOutAdr	:=  iAdrMM2AmmBase;

	xMsg1280.Num		:=	1280;
	xMsg1280.AmmInAdr	:=  iAdrAmmBase2MM;
	xMsg1280.AmmOutAdr	:=  iAdrMM2AmmBase;

	xMsg1288.Num		:=	1288;
	xMsg1288.AmmInAdr	:=  iAdrAmmBase2MM;
	xMsg1288.AmmOutAdr	:=  iAdrMM2AmmBase;

	xMsg1289.Num		:=	1289;
	xMsg1289.AmmInAdr	:=  iAdrAmmBase2MM;
	xMsg1289.AmmOutAdr	:=  iAdrMM2AmmBase;

	xMsg1290.Num		:=	1290;
	xMsg1290.AmmInAdr	:=  iAdrAmmBase2MM;
	xMsg1290.AmmOutAdr	:=  iAdrMM2AmmBase;

	xMsg1291.Num		:=	1291;
	xMsg1291.AmmInAdr	:=  iAdrAmmBase2MM;
	xMsg1291.AmmOutAdr	:=  iAdrMM2AmmBase;

	xMsg2098.Num		:=	2098;
	xMsg2098.AmmInAdr	:=  iAdrAmmBase2MM;
	xMsg2098.AmmOutAdr	:=  iAdrMM2AmmBase;

	xMsg2112.Num		:=	2112;
	xMsg2112.AmmInAdr	:=  iAdrAmmBase2MM;
	xMsg2112.AmmOutAdr	:=  iAdrMM2AmmBase;

	xMsg2113.Num		:=	2113;
	xMsg2113.AmmInAdr	:=  iAdrAmmBase2MM;
	xMsg2113.AmmOutAdr	:=  iAdrMM2AmmBase;

	xMsg2310.Num		:=	2310;
	xMsg2310.AmmInAdr	:=  iAdrAmmBase2MM;
	xMsg2310.AmmOutAdr	:=  iAdrMM2AmmBase;

	xMsg2311.Num		:=	2311;
	xMsg2311.AmmInAdr	:=  iAdrAmmBase2MM;
	xMsg2311.AmmOutAdr	:=  iAdrMM2AmmBase;

	xMsg2312.Num		:=	2312;
	xMsg2312.AmmInAdr	:=  iAdrAmmBase2MM;
	xMsg2312.AmmOutAdr	:=  iAdrMM2AmmBase;

	xMsg2313.Num		:=	2313;
	xMsg2313.AmmInAdr	:=  iAdrAmmBase2MM;
	xMsg2313.AmmOutAdr	:=  iAdrMM2AmmBase;

	xMsg2315.Num		:=	2315;
	xMsg2315.AmmInAdr	:=  iAdrAmmBase2MM;
	xMsg2315.AmmOutAdr	:=  iAdrMM2AmmBase;

	xMsg2319.Num		:=	2319;
	xMsg2319.AmmInAdr	:=  iAdrAmmBase2MM;
	xMsg2319.AmmOutAdr	:=  iAdrMM2AmmBase;

	xMsg2320.Num		:=	2320;
	xMsg2320.AmmInAdr	:=  iAdrAmmBase2MM;
	xMsg2320.AmmOutAdr	:=  iAdrMM2AmmBase;

	xMsg2321.Num		:=	2321;
	xMsg2321.AmmInAdr	:=  iAdrAmmBase2MM;
	xMsg2321.AmmOutAdr	:=  iAdrMM2AmmBase;

	xMsg2322.Num		:=	2322;
	xMsg2322.AmmInAdr	:=  iAdrAmmBase2MM;
	xMsg2322.AmmOutAdr	:=  iAdrMM2AmmBase;

	xMsg2337.Num		:=	2337;
	xMsg2337.AmmInAdr	:=  iAdrAmmBase2MM;
	xMsg2337.AmmOutAdr	:=  iAdrMM2AmmBase;

	xMsg2338.Num		:=	2338;
	xMsg2338.AmmInAdr	:=  iAdrAmmBase2MM;
	xMsg2338.AmmOutAdr	:=  iAdrMM2AmmBase;

	xMsg2340.Num		:=	2340;
	xMsg2340.AmmInAdr	:=  iAdrAmmBase2MM;
	xMsg2340.AmmOutAdr	:=  iAdrMM2AmmBase;

	xMsg2374.Num		:=	2374;
	xMsg2374.AmmInAdr	:=  iAdrAmmBase2MM;
	xMsg2374.AmmOutAdr	:=  iAdrMM2AmmBase;

	xMsg2468.Num		:=	2468;
	xMsg2468.AmmInAdr	:=  iAdrAmmBase2MM;
	xMsg2468.AmmOutAdr	:=  iAdrMM2AmmBase;

	xMsg2469.Num		:=	2469;
	xMsg2469.AmmInAdr	:=  iAdrAmmBase2MM;
	xMsg2469.AmmOutAdr	:=  iAdrMM2AmmBase;

	xMsg2494.Num		:=	2494;
	xMsg2494.AmmInAdr	:=  iAdrAmmBase2MM;
	xMsg2494.AmmOutAdr	:=  iAdrMM2AmmBase;

	xMsg2495.Num		:=	2495;
	xMsg2495.AmmInAdr	:=  iAdrAmmBase2MM;
	xMsg2495.AmmOutAdr	:=  iAdrMM2AmmBase;

	xMsg2496.Num		:=	2496;
	xMsg2496.AmmInAdr	:=  iAdrAmmBase2MM;
	xMsg2496.AmmOutAdr	:=  iAdrMM2AmmBase;

	xMsg2497.Num		:=	2497;
	xMsg2497.AmmInAdr	:=  iAdrAmmBase2MM;
	xMsg2497.AmmOutAdr	:=  iAdrMM2AmmBase;

	xMsg2498.Num		:=	2498;
	xMsg2498.AmmInAdr	:=  iAdrAmmBase2MM;
	xMsg2498.AmmOutAdr	:=  iAdrMM2AmmBase;

	xMsg2499.Num		:=	2499;
	xMsg2499.AmmInAdr	:=  iAdrAmmBase2MM;
	xMsg2499.AmmOutAdr	:=  iAdrMM2AmmBase;

	xMsg2500.Num		:=	2500;
	xMsg2500.AmmInAdr	:=  iAdrAmmBase2MM;
	xMsg2500.AmmOutAdr	:=  iAdrMM2AmmBase;

	xMsg2546.Num		:=	2546;
	xMsg2546.AmmInAdr	:=  iAdrAmmBase2MM;
	xMsg2546.AmmOutAdr	:=  iAdrMM2AmmBase;

	xMsg2547.Num		:=	2547;
	xMsg2547.AmmInAdr	:=  iAdrAmmBase2MM;
	xMsg2547.AmmOutAdr	:=  iAdrMM2AmmBase;

	xMsg2549.Num		:=	2549;
	xMsg2549.AmmInAdr	:=  iAdrAmmBase2MM;
	xMsg2549.AmmOutAdr	:=  iAdrMM2AmmBase;

	xMsg2551.Num		:=	2551;
	xMsg2551.AmmInAdr	:=  iAdrAmmBase2MM;
	xMsg2551.AmmOutAdr	:=  iAdrMM2AmmBase;

	xMsg2601.Num		:=	2601;
	xMsg2601.AmmInAdr	:=  iAdrAmmBase2MM;
	xMsg2601.AmmOutAdr	:=  iAdrMM2AmmBase;

	xMsg2622.Num		:=	2622;
	xMsg2622.AmmInAdr	:=  iAdrAmmBase2MM;
	xMsg2622.AmmOutAdr	:=  iAdrMM2AmmBase;

	xMsg2623.Num		:=	2623;
	xMsg2623.AmmInAdr	:=  iAdrAmmBase2MM;
	xMsg2623.AmmOutAdr	:=  iAdrMM2AmmBase;

	xMsg2655.Num		:=	2655;
	xMsg2655.AmmInAdr	:=  iAdrAmmBase2MM;
	xMsg2655.AmmOutAdr	:=  iAdrMM2AmmBase;

	xMsg2656.Num		:=	2656;
	xMsg2656.AmmInAdr	:=  iAdrAmmBase2MM;
	xMsg2656.AmmOutAdr	:=  iAdrMM2AmmBase;

	xMsg2657.Num		:=	2657;
	xMsg2657.AmmInAdr	:=  iAdrAmmBase2MM;
	xMsg2657.AmmOutAdr	:=  iAdrMM2AmmBase;

	xMsg2658.Num		:=	2658;
	xMsg2658.AmmInAdr	:=  iAdrAmmBase2MM;
	xMsg2658.AmmOutAdr	:=  iAdrMM2AmmBase;

	xMsg2659.Num		:=	2659;
	xMsg2659.AmmInAdr	:=  iAdrAmmBase2MM;
	xMsg2659.AmmOutAdr	:=  iAdrMM2AmmBase;

	xMsg2660.Num		:=	2660;
	xMsg2660.AmmInAdr	:=  iAdrAmmBase2MM;
	xMsg2660.AmmOutAdr	:=  iAdrMM2AmmBase;

	xMsg2661.Num		:=	2661;
	xMsg2661.AmmInAdr	:=  iAdrAmmBase2MM;
	xMsg2661.AmmOutAdr	:=  iAdrMM2AmmBase;

	xMsg2662.Num		:=	2662;
	xMsg2662.AmmInAdr	:=  iAdrAmmBase2MM;
	xMsg2662.AmmOutAdr	:=  iAdrMM2AmmBase;

	xMsg2663.Num		:=	2663;
	xMsg2663.AmmInAdr	:=  iAdrAmmBase2MM;
	xMsg2663.AmmOutAdr	:=  iAdrMM2AmmBase;

	xMsg2664.Num		:=	2664;
	xMsg2664.AmmInAdr	:=  iAdrAmmBase2MM;
	xMsg2664.AmmOutAdr	:=  iAdrMM2AmmBase;

	xMsg2743.Num		:=	2743;
	xMsg2743.AmmInAdr	:=  iAdrAmmBase2MM;
	xMsg2743.AmmOutAdr	:=  iAdrMM2AmmBase;

	xMsg2744.Num		:=	2744;
	xMsg2744.AmmInAdr	:=  iAdrAmmBase2MM;
	xMsg2744.AmmOutAdr	:=  iAdrMM2AmmBase;

	xMsg2745.Num		:=	2745;
	xMsg2745.AmmInAdr	:=  iAdrAmmBase2MM;
	xMsg2745.AmmOutAdr	:=  iAdrMM2AmmBase;

	xMsg2746.Num		:=	2746;
	xMsg2746.AmmInAdr	:=  iAdrAmmBase2MM;
	xMsg2746.AmmOutAdr	:=  iAdrMM2AmmBase;

	xMsg2747.Num		:=	2747;
	xMsg2747.AmmInAdr	:=  iAdrAmmBase2MM;
	xMsg2747.AmmOutAdr	:=  iAdrMM2AmmBase;

	xMsg2748.Num		:=	2748;
	xMsg2748.AmmInAdr	:=  iAdrAmmBase2MM;
	xMsg2748.AmmOutAdr	:=  iAdrMM2AmmBase;

	xMsg2793.Num		:=	2793;
	xMsg2793.AmmInAdr	:=  iAdrAmmBase2MM;
	xMsg2793.AmmOutAdr	:=  iAdrMM2AmmBase;

	xMsg2847.Num		:=	2847;
	xMsg2847.AmmInAdr	:=  iAdrAmmBase2MM;
	xMsg2847.AmmOutAdr	:=  iAdrMM2AmmBase;

	xMsg2848.Num		:=	2848;
	xMsg2848.AmmInAdr	:=  iAdrAmmBase2MM;
	xMsg2848.AmmOutAdr	:=  iAdrMM2AmmBase;

	xMsg3100.Num		:=	3100;
	xMsg3100.AmmInAdr	:=  iAdrAmmBase2MM;
	xMsg3100.AmmOutAdr	:=  iAdrMM2AmmBase;

	xMsg3214.Num		:=	3214;
	xMsg3214.AmmInAdr	:=  iAdrAmmBase2MM;
	xMsg3214.AmmOutAdr	:=  iAdrMM2AmmBase;

	xMsg3215.Num		:=	3215;
	xMsg3215.AmmInAdr	:=  iAdrAmmBase2MM;
	xMsg3215.AmmOutAdr	:=  iAdrMM2AmmBase;

	xMsg3313.Num		:=	3313;
	xMsg3313.AmmInAdr	:=  iAdrAmmBase2MM;
	xMsg3313.AmmOutAdr	:=  iAdrMM2AmmBase;

	xMsg3314.Num		:=	3314;
	xMsg3314.AmmInAdr	:=  iAdrAmmBase2MM;
	xMsg3314.AmmOutAdr	:=  iAdrMM2AmmBase;

	xMsg3349.Num		:=	3349;
	xMsg3349.AmmInAdr	:=  iAdrAmmBase2MM;
	xMsg3349.AmmOutAdr	:=  iAdrMM2AmmBase;

	xMsg3366.Num		:=	3366;
	xMsg3366.AmmInAdr	:=  iAdrAmmBase2MM;
	xMsg3366.AmmOutAdr	:=  iAdrMM2AmmBase;

	xMsg3394.Num		:=	3394;    (*STM*)
	xMsg3394.AmmInAdr	:=  iAdrAmmBase2MM;
	xMsg3394.AmmOutAdr	:=  iAdrMM2AmmBase;

	xMsg3395.Num		:=	3395;    (*STM*)
	xMsg3395.AmmInAdr	:=  iAdrAmmBase2MM;
	xMsg3395.AmmOutAdr	:=  iAdrMM2AmmBase;

	xMsg3397.Num		:=	3397;
	xMsg3397.AmmInAdr	:=  iAdrAmmBase2MM;
	xMsg3397.AmmOutAdr	:=  iAdrMM2AmmBase;

	xMsg3417.Num		:=	3417;
	xMsg3417.AmmInAdr	:=  iAdrAmmBase2MM;
	xMsg3417.AmmOutAdr	:=  iAdrMM2AmmBase;

	xMsg3490.Num		:=	3490;    (*STM*)
	xMsg3490.AmmInAdr	:=  iAdrAmmBase2MM;
	xMsg3490.AmmOutAdr	:=  iAdrMM2AmmBase;

	xMsg3491.Num		:=	3491;    (*STM*)
	xMsg3491.AmmInAdr	:=  iAdrAmmBase2MM;
	xMsg3491.AmmOutAdr	:=  iAdrMM2AmmBase;

	xMsg3510.Num		:=	3510;
	xMsg3510.AmmInAdr	:=  iAdrAmmBase2MM;
	xMsg3510.AmmOutAdr	:=  iAdrMM2AmmBase;

	xMsg3511.Num		:=	3511;
	xMsg3511.AmmInAdr	:=  iAdrAmmBase2MM;
	xMsg3511.AmmOutAdr	:=  iAdrMM2AmmBase;

	xMsg3512.Num		:=	3512;
	xMsg3512.AmmInAdr	:=  iAdrAmmBase2MM;
	xMsg3512.AmmOutAdr	:=  iAdrMM2AmmBase;

	xMsg3513.Num		:=	3513;
	xMsg3513.AmmInAdr	:=  iAdrAmmBase2MM;
	xMsg3513.AmmOutAdr	:=  iAdrMM2AmmBase;

	xMsg3514.Num		:=	3514;
	xMsg3514.AmmInAdr	:=  iAdrAmmBase2MM;
	xMsg3514.AmmOutAdr	:=  iAdrMM2AmmBase;

	xMsg3528.Num		:=	3528;
	xMsg3528.AmmInAdr	:=  iAdrAmmBase2MM;
	xMsg3528.AmmOutAdr	:=  iAdrMM2AmmBase;

	xMsg3580.Num		:=	3580;
	xMsg3580.AmmInAdr	:=  iAdrAmmBase2MM;
	xMsg3580.AmmOutAdr	:=  iAdrMM2AmmBase;

	xMsg3581.Num		:=	3581;
	xMsg3581.AmmInAdr	:=  iAdrAmmBase2MM;
	xMsg3581.AmmOutAdr	:=  iAdrMM2AmmBase;

	xMsg3582.Num		:=	3582;
	xMsg3582.AmmInAdr	:=  iAdrAmmBase2MM;
	xMsg3582.AmmOutAdr	:=  iAdrMM2AmmBase;

	xMsg9215.Num		:=	9215;//SWAT920/5
	xMsg9215.AmmInAdr	:=  iAdrAmmBase2MM;
	xMsg9215.AmmOutAdr	:=  iAdrMM2AmmBase;

	xMsg9249.Num		:=	9249;
	xMsg9249.AmmInAdr	:=  iAdrAmmBase2MM;
	xMsg9249.AmmOutAdr	:=  iAdrMM2AmmBase;

	xMsg9305.Num		:=	9305;
	xMsg9305.AmmInAdr	:=  iAdrAmmBase2MM;
	xMsg9305.AmmOutAdr	:=  iAdrMM2AmmBase;

	xMsg9306.Num		:=	9306;
	xMsg9306.AmmInAdr	:=  iAdrAmmBase2MM;
	xMsg9306.AmmOutAdr	:=  iAdrMM2AmmBase;

	xMsg9307.Num		:=	9307;
	xMsg9307.AmmInAdr	:=  iAdrAmmBase2MM;
	xMsg9307.AmmOutAdr	:=  iAdrMM2AmmBase;

	xMsg9308.Num		:=	9308;
	xMsg9308.AmmInAdr	:=  iAdrAmmBase2MM;
	xMsg9308.AmmOutAdr	:=  iAdrMM2AmmBase;

	xMsg9310.Num		:=	9310;
	xMsg9310.AmmInAdr	:=  iAdrAmmBase2MM;
	xMsg9310.AmmOutAdr	:=  iAdrMM2AmmBase;

	xMsg9347.Num		:=	9347;
	xMsg9347.AmmInAdr	:=  iAdrAmmBase2MM;
	xMsg9347.AmmOutAdr	:=  iAdrMM2AmmBase;

	xMsg9348.Num		:=	9348;
	xMsg9348.AmmInAdr	:=  iAdrAmmBase2MM;
	xMsg9348.AmmOutAdr	:=  iAdrMM2AmmBase;

	(* template
	xMsg.Num		:=	;
	xMsg.AmmInAdr	:=  iAdrAmmBase2MM;
	xMsg.AmmOutAdr	:=  iAdrMM2AmmBase;
	*)
END_PROGRAM
```

#### MsgEX.var
```iecst
VAR
	bNoMon4BlackStart : BOOL;
	bT_EGaHE1_LimHi_Trip : BOOL; (*STM*)
	bT_EGaHE1_LimHi_Warn : BOOL; (*STM*)
	bT_EGaHE2_LimHi_Trip : BOOL; (*STM*)
	bT_EGaHE2_LimHi_Warn : BOOL; (*STM*)
	iAdrAmmBase2MM : UDINT;
	iAdrMM2AmmBase : UDINT;
	rPr_PC_Diff : REAL;
	xGR_MAXR_Pr_Diff_ExGCoo_LimHi : GR_MAXR;
	xGR_MAXR_Pr_Diff_ExGFil_LimHi1 : GR_MAXR;
	xGR_MAXR_Pr_Diff_ExGFil_LimHi2 : GR_MAXR;
	xGR_MAXR_Pr_Diff_ExGFil_LimHiA : GR_MAXR;
	xGR_MAXR_T_EGaHE1_LimHi_Trip : GR_MAXR; (*STM*)
	xGR_MAXR_T_EGaHE1_LimHi_Warn : GR_MAXR; (*STM*)
	xGR_MAXR_T_EGaHE2_LimHi_Trip : GR_MAXR; (*STM*)
	xGR_MAXR_T_EGaHE2_LimHi_Warn : GR_MAXR; (*STM*)
	xGR_MAXR_T_EGaHE_LimHi : GR_MAXR;
	xGR_MAXR_T_EGaLPTC_A_LimHi : GR_MAXR;
	xGR_MAXR_T_EGaLPTC_B_LimHi : GR_MAXR;
	xGR_MAXR_T_EGaTC_LimHi : GR_MAXR;
	xGR_MAXR_T_EGbTC_LimHi : GR_MAXR;
	xGR_MAXR_T_EGbTC_LimHiHi : GR_MAXR;
	xGR_MAXR_T_PlateHE_LimHi : GR_MAXR;
	xGR_MAXR_T_PlateHE_LimHiHi : GR_MAXR;
	xGR_MINR_Pr_Diff_ExGFil_LimLo : GR_MINR;
	xMsg1045 : Msg;
	xMsg1046 : Msg;
	xMsg1069 : Msg;
	xMsg1092 : Msg;
	xMsg1104 : Msg;
	xMsg1106 : Msg;
	xMsg1161 : Msg;
	xMsg1162 : Msg;
	xMsg1163 : Msg;
	xMsg1164 : Msg;
	xMsg1165 : Msg;
	xMsg1169 : Msg;
	xMsg1170 : Msg;
	xMsg1171 : Msg;
	xMsg1172 : Msg;
	xMsg1173 : Msg;
	xMsg1174 : Msg;
	xMsg1273 : Msg;
	xMsg1274 : Msg;
	xMsg1275 : Msg;
	xMsg1276 : Msg;
	xMsg1277 : Msg;
	xMsg1278 : Msg;
	xMsg1279 : Msg;
	xMsg1280 : Msg;
	xMsg1288 : Msg;
	xMsg1289 : Msg;
	xMsg1290 : Msg;
	xMsg1291 : Msg;
	xMsg2098 : Msg;
	xMsg2112 : Msg;
	xMsg2113 : Msg;
	xMsg2310 : Msg;
	xMsg2311 : Msg;
	xMsg2312 : Msg;
	xMsg2313 : Msg;
	xMsg2315 : Msg;
	xMsg2319 : Msg;
	xMsg2320 : Msg;
	xMsg2321 : Msg;
	xMsg2322 : Msg;
	xMsg2337 : Msg;
	xMsg2338 : Msg;
	xMsg2340 : Msg;
	xMsg2374 : Msg;
	xMsg2468 : Msg;
	xMsg2469 : Msg;
	xMsg2494 : Msg;
	xMsg2495 : Msg;
	xMsg2496 : Msg;
	xMsg2497 : Msg;
	xMsg2498 : Msg;
	xMsg2499 : Msg;
	xMsg2500 : Msg;
	xMsg2546 : Msg;
	xMsg2547 : Msg;
	xMsg2549 : Msg;
	xMsg2551 : Msg;
	xMsg2601 : Msg;
	xMsg2622 : Msg;
	xMsg2623 : Msg;
	xMsg2655 : Msg;
	xMsg2656 : Msg;
	xMsg2657 : Msg;
	xMsg2658 : Msg;
	xMsg2659 : Msg;
	xMsg2660 : Msg;
	xMsg2661 : Msg;
	xMsg2662 : Msg;
	xMsg2663 : Msg;
	xMsg2664 : Msg;
	xMsg2743 : Msg;
	xMsg2744 : Msg;
	xMsg2745 : Msg;
	xMsg2746 : Msg;
	xMsg2747 : Msg;
	xMsg2748 : Msg;
	xMsg2793 : Msg;
	xMsg2847 : Msg;
	xMsg2848 : Msg;
	xMsg3100 : Msg;
	xMsg3214 : Msg;
	xMsg3215 : Msg;
	xMsg3313 : Msg;
	xMsg3314 : Msg;
	xMsg3349 : Msg;
	xMsg3366 : Msg;
	xMsg3394 : Msg;
	xMsg3395 : Msg;
	xMsg3397 : Msg;
	xMsg3417 : Msg;
	xMsg3490 : Msg;
	xMsg3491 : Msg;
	xMsg3510 : Msg;
	xMsg3511 : Msg;
	xMsg3512 : Msg;
	xMsg3513 : Msg;
	xMsg3514 : Msg;
	xMsg3528 : Msg;
	xMsg3580 : Msg;
	xMsg3581 : Msg;
	xMsg3582 : Msg;
	xMsg9215 : Msg; (*SWAT920/5*)
	xMsg9249 : Msg;
	xMsg9305 : Msg;
	xMsg9306 : Msg;
	xMsg9307 : Msg;
	xMsg9308 : Msg;
	xMsg9310 : Msg;
	xMsg9347 : Msg;
	xMsg9348 : Msg;
	xTOF_EngDemEPS : TOF;
	xTON_2098a : TON;
	xTON_2098b : TON;
	xTON_Pr_PC_Diff_MonRel : TON;
	xTON_9347 : TON;
END_VAR
```

### Program Logical/Exhaust/vis_EX (IEC, version 4.09.0) - visualization

#### vis_EXCyclic.st - Cyclic code
```iecst
(*******************************************************************************
vis		visualization

This code is confidential and proprietary to the INNIO Company.
It may not be used in any form, or reproduced in any manner,
without the express written permission of the INNIO Company.
Copyright, INNIO Company, 2019

Customized modifications: -
------------------------

History:
-------
V4.00.0	25.04.2012	lettenb.	new
V4.00.1	25.04.2012	lettenb.	MM2VIS.tN2_ScavSigLampOn added
V4.00.2	23.01.2015				920(stapelfeld) added
V4.03.0	29.07.2015	plattner	rPr_Diff_ExG... added
		07.08.2015  Denk		Manual operating auxiliaries control functionality added
V4.05.0	22.05.2017	TinelloM	SCR deleted
		12.07.2017	Messner		Scavenging Valve Temperature Sensor added
		04.12.2017	Messner		Oxidation catalyst added
V4.07.0	13.05.2019	lettenb.	MM2VIS.rT_EGaTC: average value to existing bus interface #505
V4.09.0	02.08.2019	lettenb.	temperature exhaust gas pressure relief valve 1/2 added
V4.14.0	16.10.2024	VighM		Fast exhaust pressure value for visualisation added

Instructions for use:
--------------------
Outstandings:
------------
*******************************************************************************)
PROGRAM _CYCLIC

	IF Para.bT_EGaLPTC_A_Active AND Para.bT_EGaLPTC_B_Active THEN
			MM2VIS.rT_EGaTC	:=  OUT_EX.rT_EGaLPTC_Avg; (* average value to existing bus interface #505 *)
	ELSE	MM2VIS.rT_EGaTC	:=	IN_EX.tT_EGaTC.Ai;
	END_IF;

	MM2VIS.rT_EGaHE			:=	IN_EX.tT_EGaHE.Ai;
	MM2VIS.rT_PlateHE		:=	IN_EX.tT_PlateHE.Ai;
	MM2VIS.rT_EGbTC			:=	IN_EX.tT_EGbTC.Ai;

	MM2VIS.rT_EGaLPTC_A		:=	IN_EX.tT_EGaLPTC_A.Ai;
	MM2VIS.rT_EGaLPTC_B		:=	IN_EX.tT_EGaLPTC_B.Ai;
	MM2VIS.rT_EGbHPTC_A		:=	IN_EX.tT_EGbHPTC_A.Ai;
	MM2VIS.rT_EGbHPTC_B		:=	IN_EX.tT_EGbHPTC_B.Ai;
	MM2VIS.rT_EGaHPTC_A		:=	IN_EX.tT_EGaHPTC_A.Ai;
	MM2VIS.rT_EGaHPTC_B		:=	IN_EX.tT_EGaHPTC_B.Ai;
	MM2VIS.rPr_EGbHPTC_A	:=	IN_EX.tPr_EGbHPTC_A.Ai;
	MM2VIS.rPr_EGbHPTC_B	:=	IN_EX.tPr_EGbHPTC_B.Ai;
	MM2VIS.rPr_EGaHPTC_A	:=	IN_EX.tPr_EGaHPTC_A.Ai;
	MM2VIS.rPr_EGaHPTC_B	:=	IN_EX.tPr_EGaHPTC_B.Ai;
	MM2VIS.rPr_EGaLPTC_A	:=	IN_EX.tPr_EGaLPTC_A.Ai;
	MM2VIS.rPr_EGaLPTC_B	:=	IN_EX.tPr_EGaLPTC_B.Ai;

	(* scavenging *)
	MM2VIS.bScavVaOpened	:=	IN_EX.tScavVaOpened.Di;
	MM2VIS.bScavFanCoOn		:=	OUT_EX.tScavFanCoOn.Do;
	MM2VIS.bN2_ScavGV_CoOpen:=	OUT_EX.tN2_ScavGV_CoOpen.Do;
	MM2VIS.bN2_ScavSigLampOn:=	OUT_EX.tN2_ScavSigLampOn.Do;
	MM2VIS.rT_bScavValve	:= 	IN_EX.tT_bScavValve.Ai;

	(* exhaust gas valves *)
	IF (IN_EX.tManAuxCtr.bGnl_Rel = TRUE) THEN
		MM2VIS.bEG_BoVaOpened	:=	IN_EX.tEG_BoVaOpened.Di;
		MM2VIS.bEG_ByVaOpened	:=	IN_EX.tEG_ByVaOpened.Di;
	ELSE
		MM2VIS.bEG_BoVaOpened	:=	OUT_EX.bEG_BoVaOpened;
		MM2VIS.bEG_ByVaOpened	:=	OUT_EX.bEG_ByVaOpened;
								Para.bEG_BoVa_Visible;	(* for vis *)
								Para.bEG_ByVa_Visible;	(* for vis *)
	END_IF;

	(* codinox *)
	MM2VIS.bCodinox_Rdy	    :=	IN_EX.tCodinox_Rdy.Di;
	MM2VIS.bCO2_VaOpened	:=	IN_EX.tCO2_VaOpened.Di;
	MM2VIS.bCO2_FanCoOn		:=	OUT_EX.tCO2_FanCoOn.Do;
	MM2VIS.bT_EGaHE1_Active	:=	Para.bCodinox_Active OR NOT Para.bT_EGaHE1_Active; (* 0=visible *)
	MM2VIS.rT_EGaHE1		:=	IN_EX.tT_EGaHE1.Ai;
	MM2VIS.bT_EGaHE2_Active	:=	Para.bCodinox_Active OR NOT Para.bT_EGaHE2_Active;
	MM2VIS.rT_EGaHE2		:=	IN_EX.tT_EGaHE2.Ai;

	MM2VIS.rPr_Diff_ExGFilter		:=	IN_EX.tPr_Diff_ExGFilter.Ai;
	MM2VIS.rPr_Diff_ExGCooler		:=  IN_EX.tPr_Diff_ExGCooler.Ai;

	(* OXIcat *)
	MM2VIS.rT_EGbCat		:= IN_EX.tT_EGbCat.Ai;
	MM2VIS.rT_EGaCat		:= IN_EX.tT_EGaCat.Ai;
	MM2VIS.rPr_OXIcat_In 	:= IN_EX.tPr_OXIcat_In.Ai;
	MM2VIS.rPr_OXIcat_Diff 	:= IN_EX.tPr_OXIcat_In.Ai - IN_EX.tPr_OXIcat_Out.Ai;

	MM2VIS.rT_EG_PrReliefVa1	:= IN_EX.tT_EG_PrReliefVa1.Ai;
	MM2VIS.rT_EG_PrReliefVa2	:= IN_EX.tT_EG_PrReliefVa2.Ai;

	(* fast exhaust pressure sensor *)
	MM2VIS.rPr_OXIcat_In_Fast := IN_EX.tPr_EG_Deflag_Fast_TC1.Ai;
END_PROGRAM
```

### Program Logical/Exhaust/ParEX (IEC, version 4.06.0) - + parameter handling

- perm_par.st (not readable text: treated as protected, skipped)

#### perm_par.var
```iecst
VAR
	tParaIntern : ParaHandler_typ; (*Connector type to perm_par*)
	tMM2ParaBase_ReadBack : MM2ParaBase_type; (*INTERNAL! V4.06 new readback structure for information from previous tasks*)
	bWriteDataObj : BOOL; (* TRUE=write data object module *)
	bDataObjLenErr : BOOL; (*Error occured in permem: data module size missmatch*)
	bCreateDataObj : BOOL; (* TRUE=create new data object *)
	bWriteOnce : BOOL; (* write permanent memory once *)
	DatObjCreate_01 : DatObjCreate; (* data object create *)
	DatObjInfoBak_02 : DatObjInfo; (* data object info *)
	DatObjDelete_01 : DatObjDelete; (* data object delete *)
	DatObjRead_01 : DatObjRead; (* data object read *)
	DatObjRead_02 : DatObjRead; (* manual initiated data object read *)
	DatObjWrite_01 : DatObjWrite; (* data object write *)
	DatObjDelete_02 : DatObjDelete; (* data object delete *)
	DatObjDelete_11 : DatObjDelete; (*Delete Backup File*)
	DatObjInfo_01 : DatObjInfo; (* data object info *)
	DatObjInfo_02 : DatObjInfo; (* data object info *)
	szModuleName : STRING[35]; (* module name of object *)
	szModuleNameBackup : STRING[35]; (* module name of posiibly created backup object *)
	DatObjCopy_01 : DatObjCopy;
	bCopyDataObj : BOOL;
	TON_WarnDelay : TON;
	TON_WritePMEM : TON; (* delay write permanent memory *)
	ulPMPointer : UDINT; (* adress of actual checksum value *)
	ulChecksum : UDINT; (* parameter checksum value *)
	pm_len : UDINT; (* permanent value lenght *)
	ulChecksumOld : UDINT; (* last vlaue of parameter checksum *)
	ulChkValue : UDINT; (* actual value of parameter pointer *)
	pm_id : UDINT; (* permanent value identifier *)
	pm_p : UDINT; (* permanent value pointer *)
	DatObjInfo_META : DatObjInfo;
	DatObjRead_META : DatObjRead;
	szMetaDataRaw : STRING[2000];
	szMetaData : ARRAY[0..4] OF STRING[35];
	szMetaDataVis : ARRAY[0..3] OF STRING[35];
	ssIndex : INT;
	ssCount : INT;
	ucMetaDataRaw : ARRAY[0..2000] OF USINT;
	ssCount2 : INT;
	szMetaDataFile : STRING[10];
	szText1 : STRING[20];
	pv_adr_IN_XX_tPB2MM : UDINT;
	pv_lng : UDINT;
	pv_lng_IN_XX_tPB2MM : UDINT;
	pv_lng_OUT_XX_tPB2MM : UDINT;
	szText2 : STRING[20];
	pv_adr_OUT_XX_tXX2PB : UDINT;
END_VAR
VAR CONSTANT
	ERR_NOERROR : UINT := 0;
END_VAR
VAR
	usPMWriteCnt : UINT;
	pm_Error : UDINT; (* permanent value error *) (* Deleted: pm : ParaMem_typ; permanent memory tags mathias, 22.8.11*)
	fun_Error : UDINT := 0; (*state > 0 = function error*)
	xLocalParaCheck : ParaCheckFUB; (*local function instance to check parameter values*)
	TON_ParaSetupOk : TON;
	bParaCheckSystemOk : BOOL;
	iDebug_ParaOkChecked : UDINT;
	bRestoreBackupDataObj : BOOL := FALSE;
	bRestoreDataObjContent : BOOL := FALSE;
	pm_id_backup : UDINT;
	pm_p_Backup : UDINT;
	DatObjCopy_02 : DatObjCopy;
	bDeleteBackupDataObj : BOOL := FALSE; (*Command to delete backup data module file on purpose*)
	bDebugPara : ARRAY[0..5] OF BOOL;
	ssIndex2 : INT;
	ssIndex3 : INT;
	ssIndex4 : INT;
	ssIndexVis : INT;
	szText : STRING[40];
	pv_adr_Para : UDINT;
	szParaSnippet : ARRAY[0..5] OF STRING[150];
	szParaIndex : STRING[10];
	slValue : DINT;
	iModuleDLD_ResetCount : INT;
	bDownloadDetected : BOOL;
	bFlagParaStructCopyWorking : BOOL; (*true, if cyclic para copying is active, 1 false cycle at every copy *)
	bStoreInitParaInDataObj : BOOL := FALSE;
	bTestflag : BOOL;
	bReadOutMETA_Once : BOOL;
	tParaCheck_iPvAdress : ARRAY[0..5] OF UDINT;
	tParaCheck_iPvLengt : ARRAY[0..5] OF UDINT;
	tParaCheck_rPvValue : ARRAY[0..5] OF REAL;
	tParaCheck_rRangeMIN : ARRAY[0..5] OF REAL;
	tParaCheck_rRangeMAX : ARRAY[0..5] OF REAL;
	tParaCheck_szPvName : ARRAY[0..5] OF STRING[35];
	ssFormatDetected : INT;
	szMetaDataPart : STRING[150];
	szFullTaskName : STRING[35];
	szFullMetaModuleName : STRING[35];
	debugLen : INT;
	debugSize : INT := 0;
	strcat_adr1 : UDINT;
	strcat_adr2 : UDINT;
	ssIndexTN : INT;
	bAlternate : BOOL;
	n : INT;
	iAlternateChecksum : DINT;
	iAlternateChecksumOld : DINT;
	ulDebugChkValue : ARRAY[0..999] OF UDINT;
	Adr1 : UDINT;
	Adr2 : UDINT;
	usPMWriteCntStepsize : UINT := 1; (*different step sizes to help debug*)
	usPMWriteCntXOR : UINT;
	usPMWriteCntAltSum : UINT;
	ulAdrPM : UDINT;
	usChkValuePM : USINT;
	ulAdrPara : UDINT;
	ulPara_len : UDINT;
	usChkValuePara : USINT;
	iDebugCountPMDifferences : DINT := 0;
	bEngineRunDetected : BOOL; (*detection status bit autocommand 100 /101  for engine run state*)
	ucMetaDataDebugInfoLine : ARRAY[0..24] OF STRING[80];
	ssIndexMand : INT := 0;
	szMetaDataMand : STRING[35];
	iMyErrorInfo_Autoreset : DINT; (*internal autoreset counter*)
	ssIndex_Version : INT; (*internal*)
	ssIndex_BU : INT; (*internal*)
	ssIndex_BU2 : INT; (*internal*)
END_VAR
```

### Program Logical/Exhaust/PermEX (IEC, version 4.07.1) - + PermanentMemory

- PermEXCyclic.st (not readable text: treated as protected, skipped)

- PermEXInit.st (not readable text: treated as protected, skipped)

#### PermEX.var
```iecst
VAR
	pm_Error : UINT;
	write_once : BOOL;
	pm_len : UDINT;
	ModulName : STRING[35];
	DatObjInfo_01 : DatObjInfo;
	pm_id : UDINT;
	pm_p : UDINT;
	bCreateDataObj : BOOL;
	perm_par_vers : UINT;
	DatObjRead_01 : DatObjRead;
	DatObjDelete_PermMem : DatObjDelete;
	DatObjCreate_01 : DatObjCreate;
	DatObjWrite_01 : DatObjWrite;
	ulChecksumOld : UDINT;
	ulPMPointer : UDINT;
	ulChkValue : UDINT;
	TON_WritePMEM : TON;
	ulChecksum : UDINT;
	bWriteDataObj : BOOL;
	TON_WarnDelay : TON;
	TON_BlockMinFileAge : TON; (*waiting time without file write after successful performed write*)
	bBlock_MinFileAge : BOOL := FALSE; (*pause the perm file write after each sucessful write*)
	iPM_WriteCnt : UDINT; (* *) (*old VarName: usPMWriteCnt*)
END_VAR
VAR CONSTANT
	ERR_NOERROR : UINT := 0;
END_VAR
VAR
	pmm : Perm_EX_Struct;
END_VAR
```

### Package Logical/Generator - GC: Generator Control

### Data object Logical/Generator/META_GC (Simple) - MODUL META data file

#### META_GC.dat
```
; *******************************************************************************
; Module Meta Data (data module)
;
; This code is confidential and proprietary to the INNIO Company.
; It may not be used in any form, or reproduced in any manner, without the express
; written permission of the INNIO Company.
; Copyright, INNIO Company, 2023
;
; Customized modifications: -
; ------------------------
;
; History:
; -------
; V3.99.00.00	06.03.2013	Weitzer,	generated for modular software
; V3.99.02.00	29.05.2013	Zengerer,	initial dependencies prepared
; V4.00.00.00	31.01.2014	Weitzer,	versions changed
; V4.01.00.00	22.07.2014	lettenb.	Para.bSyActive added
; V4.03.00.00	22.07.2014	Tinello		OilSkid added
;				15.06.2015  lettenb.	PARAMETER_CHK expanded
; V4.04.00.00	10.05.2016	lettenb.	version changed
; V4.04.00.00	12.07.2016	Zengerer 	version + dependencies changed (customer array size)
;               20.03.2017	lettenb.	DIG142: power reduct.acc.gen.air inlet temp. added-
;                                       tQ_AVR_Set_U.Ao: Q-vorgabe AVR added
; V4.04.01.00	10.07.2017	Waldhart	A2202 and A2203 disabled due to SWAT 920 # 3
; V4.05.00.00	30.11.2017	lettenb.	Q-management(GR redesign, PF control -> Q control)
; V4.05.01.00	22.02.2018	lettenb.	AI_PF_CosPCtr_Set removed
; V4.05.02.00	26.03.2018	Farre, 	 	Signals removed (PF_CosPCtr_PF1_Ena, PF_CosPCtr_PF2_Ena, PF_CosPCtr_PF3_Ena, PF_CosPCtr_PF4_Ena, PF_CosPCtr_PF5_Ena)
; V4.05.03.00	04.04.2018	lettenb.	oilskid interface: bRelEngStart_OilSkid prepared for series
; V4.05.04.00	09.04.2018	lettenb.	1036 bParaSetupOk added to avoid alarm at plc startup, bugfix
; V4.05.05.00	26.04.2018	lettenb.	SWAT920/5 added
; V4.05.06.00	10.10.2018	lettenb.	v_ctr: puls duration for voltage matching
; V4.07.00.00	11.10.2018	lettenb.	Di: tU_Gen_Inc/Dec added for diagnosis
;				24.01.2019	Schmid		A1038: IN_GC.tP_GenRev_Ext.Di / A1144: IN_GC.tI_GenAsy_Ext.Di - DIs act directly on alarms without delay
;				30.07.2019	lettenb.	LOS_Dem.Do: 1054,1031 added(safety request, doujak andreas) bu01
;										error condition for OilSkid: 1031 added, corr.for iCnt_OilSkid_HP_PrErr(safety request, doujak andreas) bu01
;				03.10.2019	lettenb.	perm data writing to CF 10s -> 10m, bu01
; V4.09.00.00	06.08.2019	lettenb.	GCB closing time measurement, Ctr_Q freeze
;				02.12.2019	lettenb.	generator protection(thaler)
; V4.10.00.00	22.05.2020	lettenb.	Eng_Bloc signales for op_state prepared
;				14.12.2020	lettenb.	TON,TOF reset added to avoid time overrun, cleanup
; V4.11.00.00	29.09.2021	lettenb.	release voltage control by customer bit added
;				25.01.2022	lettenb.	voltage droop control added(MayerR)
;				28.01.2022	Perktold	included plant controller upgrade
; V4.12.00.00	21.11.2022	lettenb.	version + dependencies
;				19.12.2022	Perktold	added comments for sr-code (EN 13849-1 / 4.6.3) for A1038
; V4.13.00.00	12.06.2023  Rimal		2371 and 2372 added, oilskid
;				04.07.2023	Perktold	A2373 and W9372 added, Earth fault protection via MMD signals
;				20.11.2023	Farre,		added IN_SY.bBypassMCB_CosPhi and request power mode interfaces from CU needed for Microgrid (2023-168)
;				07.03.2024	Farre,		issue #890, #1089: delete scaling analog input signals and shifted to HalIO
; V4.14.00.00	17.10.2024	Theobald	Alarm1112,1121,1122,1123,1124,1125,1143,1144 priority changed from 2 to 3 [2024-223]
;               25.10.2024	Farre,		Reverse power status OUT_GC.bPact_Rev to SY (2024-241)
;				18.11.2024	Farre,		enable "unbalance current monitoring A1144" based on Para.bCAsym_Ena (2024-234)
;				29.11.2024	Farre,		calculation of power reduction due to CosPhi <1, from OP to GC (issue #1700)
;
; Instructions for use:
; --------------------
; make only changes at the version numbers
; OBEY XML FORMATING RULES!
;
; Outstandings:
; ------------
;
; *******************************************************************************
;
"<META>"
;
; Module ID
"<MODUL>GC</MODUL>"
;
; Module Version (xx.yy.zz.cc)
"<VERSION>04.14.00.00</VERSION>"
;
; Module Basisupdate Version BU (00-99)
"<BASISUPDATE_VERSION>00</BASISUPDATE_VERSION>"
;
; Optional: specify order number for limitated module usage
"<ORDER></ORDER>" ;<!--(optional for restricted customizations; missing statement makes module valid for all orders)-->
;
; Parameter Check <PARAn Name='aAbcdef' MIN='xxx' MAX='yyy' />  (watch for correct spacings and apostrophs!)
"<PARAMETER_CHK>"
"<PARA1 Name='iEng_Motortype ' MIN='208' MAX='920' />"	; see general_GC for diagnosis
"<PARA2 Name='rN_EngStart_LimHi' MIN='50.0' MAX='2200.0' />"
"<PARA3 Name='rF_Nom[1] ' MIN='49' MAX='61' />"
"<PARA4 />"
"<PARA5 />"
"<PARA6 />"
"</PARAMETER_CHK>"
;
; Permanent Datamodule Filenames<!-- NAME ist ohne Dateiendung einzutragen; Nur für Counter und interne Parameter verwenden-->
"<DATAMODULES>" ;<!-- optional; mehrere DATAMODULES erlaubt-->
"	<DATAMODULE>par_GC</DATAMODULE>"
"	<DATAMODULE>perm_GC</DATAMODULE>"
"</DATAMODULES>"
;
; Dependencies Modules (MMxx.yy.zz.cc)
"<DEPENDENCIES>"
"	<DEPENDENCY MODULE='AB' VERSION='4.03.00.00' />"
"	<DEPENDENCY MODULE='AG' VERSION='4.11.00.00' />"
"	<DEPENDENCY MODULE='CH' VERSION='4.05.00.00' />"
"	<DEPENDENCY MODULE='CU' VERSION='4.13.00.00' />"
"	<DEPENDENCY MODULE='EC' VERSION='4.00.00.00' />"
"	<DEPENDENCY MODULE='EG' VERSION='4.05.00.00' />"
"	<DEPENDENCY MODULE='EX' VERSION='4.03.00.00' />"
"	<DEPENDENCY MODULE='GR' VERSION='4.05.00.00' />"
"	<DEPENDENCY MODULE='GT' VERSION='4.00.00.00' />"
"	<DEPENDENCY MODULE='HA' VERSION='4.12.00.00' />"
"	<DEPENDENCY MODULE='IG' VERSION='4.00.00.00' />"
"	<DEPENDENCY MODULE='OP' VERSION='4.10.00.00' />"
"	<DEPENDENCY MODULE='PB' VERSION='4.00.00.00' />"
"	<DEPENDENCY MODULE='SY' VERSION='4.00.00.00' />"
"   <DEPENDENCY VISVERSION='02.15.00.00' />"			; Dependencies Visualization
"</DEPENDENCIES>"
;
; Module function description
"<MODULEFUNCTION>" ;<!-- short overview documentation of module function; add reference to detailed information, if available-->
"	<General>	"
"	Generator bearing temperature, Q control, power reductions handled here. "
"	</General>	"
""
"	<F1 Name='Q-Management, AVR set point' LastModified='4.05.00.00'>"
"	Process the setpoint for the generator AVR "
"	</F1>"
"	<F2 Name='Bearing temperature monitoring and power reduction' LastModified='4.00.00.00'>"
"	Monitoring & power reduction.	"
"	</F2>"
"	<F3 Name='Generator winding temperature' LastModified='4.00.00.00'>"
"	Monitoring and power reduction.	"
"	</F3>"
"	<F4 Name='OilSkid' LastModified='4.03.00.00'>"
"	Generator bearing lubrification control	"
"	</F4>"
"	<F5 Name='OilSkid' LastModified='4.07.00.00'>"
"	Generator voltage matching.	"
"	</F5>"
""
"	<Info>"
"	Please enter additional module info here.	"
"	</Info>"
""
"	<Customized LastModified='4.00.00.00'>	"
"	- nothing "
"	</Customized>	"
""
"</MODULEFUNCTION>"
;
"</META>"
```
